(* CODESYS project BUILDING.library
   LanguageModelAttribute: qualified-access-only
   Author: OSCAT
   Version: 1.0.0.1
   Description: OSCAT Library with Building POUs.
      see ww.oscat.de for here home.
   Title: BUILDING
   DefaultNamespace: OSCAT_BUILDING
   Company: OSCAT

Project tree, tasks and I/O mapping:
  libraries: Standard, * (System); BASIC, 3.3.4.0 (OSCAT)
  Data types/
  Global Variables/
    global variables Constants
    global variables Globale_Variablen
    global variables Setup_Data
  POUs/
    actuators/
      function block ACTUATOR_2P [ST]
      function block ACTUATOR_3P [ST]
      function block ACTUATOR_A [ST]
      function block ACTUATOR_COIL [ST]
      function block ACTUATOR_PUMP [ST]
      function block ACTUATOR_UD [ST]
      function block AUTORUN [ST]
    electrical/
      function block CLICK [ST]
      function block CLICK_MODE [ST]
      function block DEBOUNCE [ST]
      function block DIMM_2 [ST]
      function block DIMM_I [ST]
      function block F_LAMP [ST]
      function block PULSE_LENGTH [ST]
      function block PULSE_T [ST]
      function block SW_RECONFIG [ST]
      function block SWITCH_I [ST]
      function block SWITCH_X [ST]
      function block TIMER_1 [ST]
      function block TIMER_2 [ST]
      function TIMER_EVENT_DECODE [ST]
      function block TIMER_EXT [ST]
      function block TIMER_P4 [ST]
    HLK/
      function AIR_DENSITY [ST]
      function AIR_ENTHALPY [ST]
      function block BOILER [ST]
      function block BURNER [ST]
      function DEW_CON [ST]
      function DEW_RH [ST]
      function DEW_TEMP [ST]
      function HEAT_INDEX [ST]
      function block HEAT_METER [ST]
      function block HEAT_TEMP [ST]
      function block LEGIONELLA [ST]
      function SDD [ST]
      function SDD_NH3 [ST]
      function SDT_NH3 [ST]
      function block T_AVG24 [ST]
      function block TANK_LEVEL [ST]
      function TANK_VOL1 [ST]
      function TANK_VOL2 [ST]
      function block TEMP_EXT [ST]
      function WATER_CP [ST]
      function WATER_DENSITY [ST]
      function WATER_ENTHALPY [ST]
      function WCT [ST]
    Jalousie/
      function block BLIND_ACTUATOR [ST]
      function block BLIND_CONTROL [ST]
      function block BLIND_CONTROL_S [ST]
      function block BLIND_INPUT [ST]
      function block BLIND_NIGHT [ST]
      function block BLIND_SCENE [ST]
      function block BLIND_SECURITY [ST]
      function block BLIND_SET [ST]
      function block BLIND_SHADE [ST]
      function block BLIND_SHADE_S [ST]
      function block BLIND_MASTER_CONECTOR [ST]
    Other/
      function BUILDING_VERSION [ST]
  Visualizations/
  global variables PersistentVars
  Documentation/
    oscat-building100-en
    oscat_building100_de
  00000000-0000-0000-0000-000000000000|D:\src\CODESYS Store\OSCAT\OSCAT_Building\trunk\Documents\Documentation\oscat_building100_de.pdf
  00000000-0000-0000-0000-000000000000|C:\Users\e.schwellinger\Desktop\oscat-building100-en.pdf
*)

// Global Variables/Constants
VAR_GLOBAL CONSTANT
END_VAR

// Global Variables/Globale_Variablen
VAR_GLOBAL
END_VAR

// PersistentVars
VAR_GLOBAL PERSISTENT RETAIN
END_VAR

// Global Variables/Setup_Data
VAR_GLOBAL RETAIN

END_VAR

// POUs/actuators/ACTUATOR_2P
FUNCTION_BLOCK ACTUATOR_2P
VAR_INPUT
	IN : BYTE;
	TEST : BOOL;
	ARE : BOOL := TRUE;
END_VAR
VAR_IN_OUT
	ARX : BOOL;
END_VAR
VAR_INPUT CONSTANT
	CYCLE_TIME : TIME;
	SENS : BYTE;
	SELF_ACT_TIME : TIME;
	SELF_ACT_PULSE : TIME;
	SELF_ACT_CYCLES : INT := 1;
END_VAR
VAR_OUTPUT
	OUT : BOOL;
	ARO : BOOL;
END_VAR
VAR
	timer : AUTORUN;
	pwgen : OSCAT_BASIC.GEN_PULSE;
END_VAR


(*
version 2.1	24. jan. 2009
programmer 	hugo
tested by		oscat

this is an intelligent actuator interface for any 2point actuator like coil drive.
the 2Point actuator can only switch on/off and therefore the input must be converted to on/off cycles.
the interface can be programmed with double click on the symbol.
in addition a self_act_time and self_act_cycles ca be programmed to switch n times on/off every self_act_time to avoid a valve to freeze.
the input value must be between 0 and 255. with the setup variable sens one can specify what must be the minimum input to turn the valve on at all.
at the same time an input > 255-sens will turn the valve on at all times.


*)

(* run the autorun timer *)
timer(trun := SELF_ACT_PULSE * (2 * SELF_ACT_CYCLES), toff := SELF_ACT_TIME, Test := TEST, ARE := ARE, arx := ARX);
ARO := timer.ARO;

(* run the pulse width generator *)
IF aro THEN
	pwgen(PTL := SELF_ACT_PULSE, PTH := SELF_ACT_PULSE);
	out := pwgen.Q;
ELSIF in < sens THEN
	out := FALSE;
ELSIF in > BYTE#255 - sens THEN
	out := TRUE;
ELSE
	pwgen.PTH := (CYCLE_TIME * OSCAT_BASIC.BAND_B(IN,SENS)) / 255;
	pwgen.PTL := CYCLE_TIME - pwgen.PTH;
	pwgen();
	out := pwgen.Q;
END_IF;



(* revision history
hm	7.10.2006 		rev 1.1
	changed error pos could not reach 1 or 0 under certain conditions due to error in code.
	changed on and off in force and force_in for better usability.

hm	17.1.2007		rev 1.2
	deleted unused variable time_overflow

hm	15.9.2007		rev 1.3
	replaced time() with T_PLC_MS for compatibility and performance reasons

hm	19. 11 2007		rev 1.4
	replaced left over statement time() with tx

hm	27. 12. 2007	REV 1.5
	CHANGED CODE FOR BETTER PERFORMANCE

hm	21. oct. 2008	rev 1.6
	code optimized

hm	23. nov. 2008	rev 2.0
	new code using library modules

hm	24. jan. 2009	rev 2.1
	deleted unused var inb
*)

END_FUNCTION_BLOCK

// POUs/actuators/AUTORUN
FUNCTION_BLOCK AUTORUN
VAR_INPUT
	IN : BOOL;
	TEST : BOOL;
	ARE : BOOL := TRUE;
END_VAR
VAR_IN_OUT
	ARX : BOOL;
END_VAR
VAR_INPUT CONSTANT
	TRUN : TIME;
	TOFF : TIME;
END_VAR
VAR_OUTPUT
	OUT : BOOL;
	ARO : BOOL;
END_VAR
VAR
	timer : OSCAT_BASIC._RMP_B;
	val : BYTE;
END_VAR



(*
version 1.0	20. nov 2008
programmer 	hugo
tested by	oscat




*)

(* run the integrator when T_off > T#0s *)
IF TOFF > T#0s THEN
	timer(DIR:= OUT, TR := SEL(OUT, TOFF, TRUN), RMP := val);
ELSE
	val := 255;
END_IF;


(* when timer = 0 or test then initiate autorun until timer reaches 255 *)
IF (NOT ARX AND ARE AND val = 0) OR TEST THEN
	val := 0;
	ARO := TRUE;
	ARX := TRUE;
ELSIF val = 255 AND ARO THEN
	ARO := FALSE;
	ARX := FALSE;
END_IF;

(* output is true when autorun ARO is true or in = TRUE *)
out := IN OR ARO;



(* revision history
hm 20. nov. 2008	rev 1.0
	original version

*)

END_FUNCTION_BLOCK

// POUs/electrical/CLICK
FUNCTION_BLOCK CLICK
VAR_INPUT
	in : BOOL;
END_VAR
VAR_OUTPUT
	Q : BOOL;
	single : BOOL;
	double : BOOL;
	triple : BOOL;
	status: BYTE;
END_VAR
VAR_INPUT CONSTANT
	T_debounce : TIME := t#10ms;
	T_short : TIME := t#200ms;
	T_pause : TIME := t#500ms;
	T_reconfig : TIME := t#1m;
END_VAR
VAR
	s_in : SW_RECONFIG;
	tx: TIME;
	state: INT;
	last: TIME;
END_VAR

(*
version 2.0	28. dec. 2008
programmer 	oscat
tested by		oscat

click checks an input for single, double or tripple click and sets the corresponding output single, doulbe or triple for the time the input stays high at the last click.
the maximum high and low time for a click can be configured with setup variables.
the input configures itself to be high or low active depending on which state the input stays longer than t_reconfig.

*)

(* reconfiguration and debounce circuitry *)
s_in(in := in, TD := T_debounce, TR := T_reconfig);

(* read system time *)
tx := DWORD_TO_TIME(OSCAT_BASIC.T_PLC_MS());

(* count the mumber of clicks *)
IF s_in.Q XOR Q THEN
	last := tx;
	IF s_in.Q THEN state := state + 1; END_IF;
END_IF;
Q := s_in.Q;

(* set outputs *)
IF state > 0 THEN
	IF (Q AND tx - last > t_short) OR (NOT Q AND tx - last > t_pause) THEN
		CASE state OF
			1:	single := TRUE;
				status := 111;
			2:	double := TRUE;
				status := 112;
			3:	triple := TRUE;
				status := 113;
		END_CASE;
		state := 0;
	END_IF;
ELSIF NOT q THEN
	single := FALSE;
	double := FALSE;
	triple := FALSE;
	status := 110;
	last := tx;
	state := 0;
END_IF;





(* revision history

15 Feb 2007	rev 1.0	hm
	created original version

18.5.2007	rev 1.1 hm
	corrected an error while execution would stop after t_reconfig elapsed.

15.9.2007	rev 1.2 hm
	replaced Time() with T_PLC_MS for compatibility and performance reasons

28. dec. 2008	rev 2.0
	rewritten using modular approach

*)

END_FUNCTION_BLOCK

// POUs/electrical/DEBOUNCE
FUNCTION_BLOCK DEBOUNCE
VAR_INPUT
	IN : BOOL;
	TD : TIME;
	PM : BOOL;
END_VAR

VAR_OUTPUT
	Q : BOOL;
END_VAR
VAR
	deb : OSCAT_BASIC.TOF;
END_VAR

(*
version 1.0	22. sep. 2008
programmer 	oscat
tested by	tobias

DEBOUNCE is used to debounce switch inputs.
in addition to the debounce functionality this FB can also be used to detect rising edges on IN when PM = TRUE.
When PM = FALSE, Q follows in with the debounce functionality.

*)


IF NOT deb.Q AND IN THEN
	(* rising edge on input detetced a *)
	Q := TRUE;
ELSIF NOT PM THEN
	Q := deb.Q;
ELSE
	Q := FALSE;
END_IF;

(* run debounce timer *)
deb(IN := IN, PT := TD);



(*
hm 22. sep. 2008	rev 1.0
	original version

*)

END_FUNCTION_BLOCK

// POUs/electrical/SW_RECONFIG
FUNCTION_BLOCK SW_RECONFIG
VAR_INPUT
	IN : BOOL;
	TD : TIME;
	TR : TIME;
END_VAR
VAR_OUTPUT
	Q : BOOL;
END_VAR
VAR
	T1, T2 : OSCAT_BASIC.TON;
	INV: BOOL;
END_VAR


(*
version 1.0	22. oct. 2008
programmer 	hugo
tested by	oscat

SW_reconfig detects if an input is high or low active and debounces the input

*)

(* run debounce circuit *)
t1(in := IN, PT := TD);

IF tr > t#0s THEN
	(* generate output *)
	Q := t1.Q XOR inv;
	(* reconfiguration timer *)
	T2(in := Q, pt := TR);
	(* when T2.Q goes high then reverse INV *)
	IF T2.Q THEN INV := NOT INV; END_IF;
ELSE
	Q := t1.Q;
END_IF;



(* revision history
hm	22.10.2008	rev 1.0
	original version

*)

END_FUNCTION_BLOCK

// POUs/actuators/ACTUATOR_3P
FUNCTION_BLOCK ACTUATOR_3P
VAR_INPUT
	IN : BYTE;
	TEST : BOOL;
	ARE : BOOL := TRUE;
	END_POS : BOOL;
END_VAR
VAR_INPUT CONSTANT
	T_RUN : TIME := t#60s;
	T_EXT : TIME := T#10s;
	T_CAL : TIME := t#600s;
	T_DIAG : TIME := T#10d;
	SWITCH_AVAIL : BOOL;
END_VAR
VAR_IN_OUT
	ARX : BOOL;
END_VAR
VAR_OUTPUT
	OUT1 : BOOL;
	OUT2 : BOOL;
	POS : BYTE;
	ERROR : BOOL;
	STATUS : BYTE;
END_VAR
VAR
	ramp : OSCAT_BASIC._RMP_NEXT;
	tx : TIME ;
	next_cal : TIME;
	next_diag : TIME;
	last: TIME;
	start: TIME;
END_VAR


(*
version 2.0	28. jan 2010
programmer 	hugo
tested by		oscat

actuator_3P is an interface for a 3 point actuator.
a 3P actuator is a motor with 2 directions that drives a valve or flap. the position of the valve or flap is controlled by runtime of the motor foreward or backward.
the available inputs are:
IN specifies the position of the actuator, 0 = 0% and 255 = 100%.
an END_POS input is available for an end_pos switch, this switch indicates the valve or flap to be at either 0% or 100%
a TEST input can at any time start a diag cycle which turns the motor towards the 0% position, then measures the runtime to 100% and then the runtime to 0%
these runtimes are stored and used for absolute positioning of the motor during normal operation. this feature is only avaliable with an END_POS switch connected to the input.
a setup variable T_DIAG can be used to specify how often the actuator repeates this auto_diag cycle automatically.
at power on a diag cycle is perfomed automatically.
a time of 0 for T_DIAG means auto diag is never performed.

the outputs out1 and out2 are for the two directions of the motor.
a pos output indicates the simulated position of the actuator during operation.
a error output is activated when the specified max_runtime is reached by any direction during debug without an end_switch to become active.
also when the up and down direction differs by more then 10% the error output is set.

for absolute positioning accuracy the actuator has a setup variable "cal_runtime" if this is set the actuator measures the total runtime of the motors and when this 
cal_runtime is exceeded it resets the actuator to 0% position and sets the output again to assure absolute accuracy.

test and calibration can be shut off by setting the appropriate values to 0.
a switch_available setup variable specifies if end_pos switches are available.

*)

(* read system timer *)
tx := DWORD_TO_TIME(OSCAT_BASIC.T_PLC_MS());

(* check test input *)
IF TEST THEN
	status := 103;
	start := tx;
	ARX := TRUE;
END_IF;

CASE status OF
	0:	(* power on setup *)
		IF ARE AND NOT ARX THEN
			status := 103;
			start := tx;
			ARX := TRUE;
		END_IF;

	100:	(* normal operation *)
		(* check for auto diagnostics *)
		IF T_DIAG > T#0s AND tx > next_diag AND ARE AND NOT ARX THEN
				status := 103;
				start := tx;
				ARX := TRUE;

		(* check for auto calibration *)
		ELSIF T_CAL > T#0s AND tx > next_cal AND ARE AND NOT ARX THEN
			IF pos > BYTE#127 THEN
				OUT1 := TRUE;
				OUT2 := FALSE;
				ramp.IN := 255;
				ARX := TRUE;
			ELSE
				OUT1 := FALSE;
				OUT2 := TRUE;
				ramp.IN := 0;
				ARX := TRUE;
			END_IF;
			status := 101;
			start := tx;
		ELSE
			(* increment next_cal if not active *)
			IF NOT(OUT1 OR OUT2) THEN next_cal := next_cal + (tx-last); END_IF;
			(* set ramp generator to IN *)
			ramp.IN := IN;
		END_IF;

	101:	(* calibrate *)
		IF tx - start < T_EXT THEN
			next_cal := tx + T_CAL;
		ELSIF SWITCH_AVAIL AND END_POS THEN
			STATUS := 100;
			ARX := FALSE;
		ELSIF tx - start > T_EXT + T_RUN THEN
			ERROR := SWITCH_AVAIL;
			ARX := FALSE;
		END_IF;

	103:	(* diagnostics up*)
		(* run up for T_ext *)
		IF tx - start < T_EXT THEN
			ERROR := FALSE;
			ramp.TR := T_RUN;
			ramp.TF := T_RUN;
			OUT1 := TRUE;
			OUT2 := FALSE;
			ramp.IN := 255;
		ELSIF SWITCH_AVAIL AND END_POS THEN
			ramp.TR := tx - start;
			STATUS := 104;
		ELSIF tx - start > T_EXT + T_RUN THEN
			ERROR := SWITCH_AVAIL;
			STATUS := 104;
			start := tx;
		END_IF;

	104:	(* diagnostics dn*)
		IF tx - start < T_ext THEN
			OUT1 := FALSE;
			OUT2 := TRUE;
			ramp.IN := 0;
			next_diag := tx + T_DIAG;
		ELSIF SWITCH_AVAIL AND END_POS THEN
			ramp.TR := tx - start;
			(* check if runtimes differ by more than 10% *)
			IF DINT_TO_TIME(ABS(TIME_TO_DINT(ramp.TR) - TIME_TO_DINT(ramp.TF))*10) > T_RUN THEN error := TRUE; END_IF;
			STATUS := 100;
			ARX := FALSE;
			next_cal := tx + T_CAL;
		ELSIF tx - start > T_EXT + T_RUN THEN
			IF SWITCH_AVAIL THEN ERROR := TRUE; END_IF;
			STATUS := 100;
			ARX := FALSE;
			next_CAL := tx + T_CAL;
		END_IF;
END_CASE;

(* internal flap simulation and output activation *)
ramp(OUT := POS);
IF STATUS = 100 THEN
	OUT1 := ramp.UP;
	OUT2 := ramp.DN;
END_IF;

(* adjust position if end switch is active *)
IF SWITCH_AVAIL AND END_POS THEN
	POS := SEL(POS > 127, 0, 255);
	next_cal := tx + T_CAL;
END_IF;

(* set last to tx for next cycle *)
last := tx;



(* revision history

hm	19. oct 2006	rev 1.1
	added security checks for end_switch to avoid overrun of the end_switch, hans

hm	23. jan 2007	rev 1.2
	deleted unused variables force_on and force_off

hm	15. sep 2007	 rev 1.3
	replaced Time() with T_PLC_MS for compatibility and performance reasons

hm	28. jan 2010	rev 2.0
	new code and new features

*)

END_FUNCTION_BLOCK

// POUs/actuators/ACTUATOR_A
FUNCTION_BLOCK ACTUATOR_A
VAR_INPUT
	I1 : BYTE;
	IS : BOOL;
	I2 : BYTE;
	RV : BOOL;
	DX : BOOL;
END_VAR
VAR_INPUT CONSTANT
	RUNTIME : TIME;
	SELF_ACT_TIME : TIME;
	OUT_MIN : WORD;
	OUT_MAX : WORD;
END_VAR
VAR_OUTPUT
	Y : WORD;
END_VAR
VAR
	timer : OSCAT_BASIC.CYCLE_4;
	dx_edge: BOOL;
END_VAR


(*
version 1.0 8. nov. 2008	
programmer 	hugo
tested by	oscat

ACTUATOR_A drives any valve or similar with 0 - 255 continuous control input.
 
*)

(* run the system timer, if self_act_time = t#0s then state is set to 0 *)
timer(T0 := RUNTIME, T1 := RUNTIME, T3 := SELF_ACT_TIME, sl := DX AND NOT dx_edge, sx := 0, S0 := SELF_ACT_TIME > t#0s);
dx_edge := dx;

CASE timer.STATE OF
	0: 	(* self act min value *)
		Y := OUT_MIN;
	1:	(* self_act max value *)
		Y := OUT_MAX;
	3:	(* normal operation *)
		IF rv THEN
			Y := OUT_MAX - (OUT_MAX - OUT_MIN) * SEL(IS, I1, I2) / 255;
		ELSE
			Y := (OUT_MAX - OUT_MIN) * SEL(IS, I1, I2) / 255 + OUT_MIN;
		END_IF;
END_CASE;




(*
hm 	8. nov. 2008	rev 1.0
	original version

*)

END_FUNCTION_BLOCK

// POUs/actuators/ACTUATOR_COIL
FUNCTION_BLOCK ACTUATOR_COIL
VAR_INPUT
	IN : BOOL;
END_VAR
VAR_INPUT CONSTANT
	self_act_cycle : TIME := t#10d;
	self_act_time : TIME := t#1s;
END_VAR
VAR_OUTPUT
	OUT :BOOL;
	STATUS : BYTE;
END_VAR
VAR
	last : DWORD;
	init: BOOL;
	tx: DWORD;
	now: DWORD;
END_VAR


(*
version 1.0	1. jun. 2008
programmer 	hugo
tested by		tobias

this is an intelligent actuator interface for any coil actuator.
the coil actuator can only switch on/off.
coil actuators like vents can get stuck if they are not u8sed for a long time and need to be autoactivated on ce in a while.

*)

(* read system time *)
now := OSCAT_BASIC.T_PLC_MS();

(* initialize for first cycle *)
IF NOT init THEN
	last := now;
	init := TRUE;
ELSIF IN THEN
	OUT := TRUE;
	STATUS := 101; (* activated by input *)
	LAST := now;
ELSE
	OUT := FALSE;
	STATUS := 100; (* disabled *)
	(* now we need to check for self activation *)
	tx := now - last;
	IF (self_act_cycle > T#0s) AND (tx >= TIME_TO_DWORD(self_act_cycle)) THEN
		OUT := TRUE;
		STATUS := 102; (* auto activation *)
		IF tx >= TIME_TO_DWORD(self_act_cycle + self_act_time) THEN
			last := now;
			OUT := FALSE;
			STATUS := 100; (* idle *)
		END_IF;
	END_IF;
END_IF;



(*
revision history:

hm		1. jun. 2008 	rev 1.0
	original version

*)

END_FUNCTION_BLOCK

// POUs/actuators/ACTUATOR_PUMP
FUNCTION_BLOCK ACTUATOR_PUMP
VAR_INPUT
	IN : BOOL;
	MANUAL : BOOL;
	RST : BOOL;
END_VAR
VAR_INPUT CONSTANT
	MIN_ONTIME : TIME := t#10s;
	MIN_OFFTIME : TIME := t#10s;
	RUN_EVERY : TIME := t#10000m;
END_VAR
VAR_OUTPUT
	PUMP : BOOL;
END_VAR
VAR_IN_OUT
	RUNTIME : UDINT;
	CYCLES : UDINT;
END_VAR
VAR
	tx : TIME;
	last_change : TIME;
	meter : OSCAT_BASIC.ontime;
	old_man : BOOL;
	init: BOOL;
END_VAR

(*
version 1.4		21. oct. 2008
programmer 		oscat
tested BY		oscat

actuator_pump is a pump interface which can be controlled by an input in and an input manual.
in or manual high turns the pump output on.
a rst input is used to reset the runtime counters.
when the pump was not active for a time run_every the actuator turns on the pump automatically for min_ontime.
two setup variables min_ontime and min_offtime guarantee a minimum runtime and offtime of the pump.
the units are hours and the output type is real to prevent from overfow.

*)

tx := DWORD_TO_TIME(OSCAT_BASIC.T_PLC_MS());

IF NOT init THEN
	init := TRUE;
	last_change := tx;
ELSIF rst THEN
	rst := FALSE;
	runtime := 0;
	cycles := 0;
ELSIF manual AND NOT pump AND NOT old_man THEN
	last_change := tx;
	pump := TRUE;
ELSIF NOT manual AND old_man AND pump AND NOT in THEN
	last_change := tx;
	pump := FALSE;
ELSIF in AND NOT pump AND tx - last_change >= min_offtime THEN
	last_change := tx;
	pump := TRUE;
ELSIF pump AND NOT in AND NOT manual AND tx - last_change >= min_ontime THEN
	last_change := tx;
	pump := FALSE;
ELSIF NOT pump AND (tx - last_change >= run_every) AND (run_every > T#0s) THEN
	last_change := tx;
	pump := TRUE;
END_IF;

meter(in := pump, seconds := runtime, cycles := cycles);
old_man := manual;



(*
hm	27.12.2006		rev 1.1
	fixed a failure while the pump would run for tmin after startup.

hm	15.9.2007		rev 1.2
	replaced Time() with T_PLC_MS for compatibility and performance reasons

hm	13. oct. 2008	rev 1.3
	auto activation can now be disabled when run_every = t#0s

hm	21. oct. 2008	rev 1.4
	changed to use ontime rev 2.0

*)

END_FUNCTION_BLOCK

// POUs/actuators/ACTUATOR_UD
FUNCTION_BLOCK ACTUATOR_UD
VAR_INPUT
	UD : BOOL;
	ON : BOOL;
	Manual : BOOL;
	Up : BOOL;
	Dn : BOOL;
	off : BOOL;
	YUP_in : BOOL;
	YDN_in : BOOL;
END_VAR
VAR_INPUT CONSTANT
	TON : TIME;
	TOFF : TIME;
	out_return : BOOL;
END_VAR
VAR_OUTPUT
	Yup : BOOL;
	Ydn : BOOL;
	status : BYTE;
END_VAR
VAR
	tx : TIME;
	last : TIME;
	init: BOOL;
END_VAR

(*
version 1.3	17. oct. 2008
programmer 	hugo
tested by		tobias

out_ud is a up/dn or Right/left locked output driver.
it can be controlled by automatic inputs UD and ON as well as manual inputs for up and dn.
a security input to shut off at any time is prvided by the off input.
two time set inputs ton and toff specify a minimum on time for outputs and a minimum off time before the next output can become active.
the module assures that only one output can be active at any time.
for higher security pls make sure you use hardware locking of the outputs to prevent from defective wiring or outputs.
further security is provided b feedback inputs Yup_in and Ydn_in which are separate inputs for the output signal, if these inputs are not available 
pls connect them directly to Yup and Ydn.
manual mode will override automatic mode by setting the manual input high.
a status output will be 0 for normal operation or 1 - 99 for error reporting and 101 - 199 for status reporting
The status output is ESR comptible.
*)

(* read system time *)
tx := DWORD_TO_TIME(OSCAT_BASIC.T_PLC_MS());

IF NOT init THEN
	(* INITIALIZATION AT FIRST CALL *)
	last := tx;
	init := TRUE;
ELSIF off THEN
	(* emergency shut off detected *)
	Yup := FALSE;
	ydn := FALSE;
	last := tx;
	status := 101;

(* Watch FOR MIN TON TIME *)
ELSIF ((Yup OR Ydn) AND tx - last < Ton) THEN
	RETURN;
ELSIF NOT yup AND NOT ydn AND tx - last < toff THEN
	RETURN;

(* manual operation *)
ELSIF manual THEN
	status := 102;
	(* directional chage set both outs 0 first *)
	IF yup AND NOT up OR ydn AND NOT dn THEN
		ydn := FALSE;
		yup := FALSE;
		last := tx;
	(* manual up operation *)
	ELSIF UP AND NOT DN AND NOT OFF THEN
		Ydn := FALSE;
		Yup := TRUE;
		last := tx;
		status := 103;
	(* manual down operation *)
	ELSIF DN AND NOT UP AND NOT OFF THEN
		Yup := FALSE;
		Ydn := TRUE;
		last := tx;
		status := 104;
	(* maual mode but no up or down *)
	ELSE
		IF YUP OR YDN THEN LAST := tx; END_IF;
		Yup := FALSE;
		ydn := FALSE;
	END_IF;

(* automatic operation *)
ELSE
	(* directional change set outputs low first *)
	IF yup AND NOT ud OR ydn AND UD THEN
		yup := FALSE;
		ydn := FALSE;
		last := tx;
	(* automatic up operation *)
	ELSIF Ud AND on AND NOT OFF THEN
		Ydn := FALSE;
		Yup := TRUE;
		last := tx;
		status := 111;

	(* automatic down operation *)
	ELSIF NOT UD AND on AND NOT OFF THEN
		Yup := FALSE;
		Ydn := TRUE;
		last := tx;
		status := 112;
	(* standby mode *)
	ELSE
		IF Yup OR Ydn THEN last := tx; END_IF;
		Yup := FALSE;
		Ydn := FALSE;
		status := 110;
	END_IF;
END_IF;

(* make sure Yup and Ydn are never on at the same time *)
IF Ydn AND Yup_in AND out_return THEN
	Ydn := FALSE;
	status := 1;
END_IF;
IF Yup AND Ydn_in AND out_return THEN
	Yup := FALSE;
	status := 2;
END_IF;



(* revision history
hm 22. jan 2007	rev 1.1
	added status output
	changed inputs ton, toff to config variables
	added config var out_return to enable yup_in and Ydn_in
	manual mod will override automatic mode 

hm	15.9.2007	rev 1.2
	replaced Time() with T_PLC_MS for compatibility and performance reasons

hm	17. oct. 2008	rev 1.3
	deleted unnecessary initialization with 0
*)

END_FUNCTION_BLOCK

// POUs/HLK/AIR_DENSITY
FUNCTION AIR_DENSITY : REAL
VAR_INPUT
	T : REAL;
	P : REAL;
	RH : REAL;
END_VAR
VAR CONSTANT
	RL : REAL := 287.05;
	RX : REAL := 3.773319E-3;
END_VAR


(*
version 1.3	13. mar. 2009
programmer 	hugo
tested by		tobias

this function calculates the air density between 0 and 100 deg C

*)

AIR_DENSITY := OSCAT_BASIC.phys.PN * (1.0 - RH * SDD(T, TRUE) * RX / P) / (RL * ( T - OSCAT_BASIC.phys.T0));

(* original code used for rev 1.0

SDD := SDD(T,FALSE);
RF := RL / (1- RH*SDD/P*RX);
Air_density := P / (RF * (T-TK));

*)

(* revision history

hm	29.10.2007	rev 1.0
	original version

hm	4.12.2007		rev 1.1
	changed code for better performance

hm	18. oct. 2008	rev 1.2
	using phys constants

hm	13. mar. 2009	rev 1.3
	real constants updated to new systax using dot

*)

END_FUNCTION

// POUs/HLK/SDD
FUNCTION SDD : REAL
VAR_INPUT
	T : REAL;
	ICE: BOOL;
END_VAR


(*
version 1.1	2 dec 2007
programmer 	hugo
tested by		tobias

this function calculates the vapor saturation pressure for moist Air over ice or water

*)

IF ice THEN
	SDD := 611.153 * EXP(22.4433 * T / (272.186 + T));
ELSE
	SDD := 611.213 * EXP(17.5043 * T / (241.2 + T));
END_IF;



(* revision history

hm 29 oct 2007		rev 1.0
	original version

hm	2. dec 2007		rev 1.1
	changed code for better performance
*)

END_FUNCTION

// POUs/HLK/AIR_ENTHALPY
FUNCTION AIR_ENTHALPY : REAL
VAR_INPUT
	T : REAL;
	RH : REAL;
END_VAR
VAR CONSTANT
	CPL : REAL := 1.00482;
	CW : REAL := 1.86;
	LH : REAL := 2500.78;
END_VAR


(*
version 1.1	2 nov 2007
programmer 	hugo
tested by		tobias

this function calculates the enthalpy for humid air between 0 and 100 deg C

*)

AIR_ENTHALPY := CPL * T + (CW * T + LH) * DEW_CON(RH,T);

(* revision history

hm	31.10.2007	rev 1.0
	original version

hm	2.11.2007		rev 1.1
	deleted unused variable RF

hm	2.12.2007		rev 1.2
	changed code for better performance
*)

END_FUNCTION

// POUs/HLK/DEW_CON
FUNCTION DEW_CON : REAL
VAR_INPUT
	RH : REAL;
	T : REAL;
END_VAR


(*
version 1.6	19. jan. 2011
programmer 	hugo
tested by		oscat

this function calculates the water concentratin in air for a given temperature and relative humidity.
the output states the concentration of water vapor in air in Gramms / qubic meter.

*)

(*	this code is good to read but need to be improoved
	SDD := 6.1078*EXPT(10,(a*T)/(b+T));
	DD := RH/100 * SDD;
	V := LOG(DD/6.1078);
	TD := b*V/(a-v);
	dew_con := 0.1 * mw / RU * DD / (T - TK);
*)
IF RH > 0.0 AND T > -50.0 THEN
	DEW_CON := 2.166824303E-2 * RH * SDD(T,FALSE)  / (T - OSCAT_BASIC.phys.T0);
ELSE
	DEW_CON := 0.0;
END_IF;

(*
Bezeichnungen:
r = relative Luftfeuchte
T = Temperatur in °C
TK = Temperatur in Kelvin (TK = T + 273.15)
TD = Taupunkttemperatur in °C
DD = Dampfdruck in hPa
SDD = Sättigungsdampfdruck in hPa

Parameter:
a = 7.5, b = 237.3 für T >= 0
a = 7.6, b = 240.7 für T < 0 über Wasser (Taupunkt)
a = 9.5, b = 265.5 für T < 0 über Eis (Frostpunkt)

R* = 8314.3 J/(kmol*K) (universelle Gaskonstante)
mw = 18.016 kg (Molekulargewicht des Wasserdampfes)
AF = absolute Feuchte in g Wasserdampf pro m3 Luft

Formeln:

   1. SDD(T) = 6.1078 * 10^((a*T)/(b+T))
   2. DD(r,T) = r/100 * SDD(T)
   3. r(T,TD) = 100 * SDD(TD) / SDD(T)
   4. TD(r,T) = b*v/(a-v) mit v(r,T) = log10(DD(r,T)/6.1078)
   5. AF(r,TK) = 10^5 * mw/R* * DD(r,T)/TK; AF(TD,TK) = 10^5 * mw/R* * SDD(TD)/TK 

*)

(* revision history

hm 29 apr 2007	rev 1.0
	original version

hm	13.sep 2007	rev 1.1
	improoved coding for speed
	deleted unused variabled SDD,DD,V, TD

hm	2. dec 2007	rev 1.2
	changed code for better performance
	output is now in Gramms / Qubic meter

hm	14. oct. 2008	rev 1.3
	performance improvement

hm	18. oct. 2008	rev 1.4
	using phys constants

hm	13. mar. 2009	rev 1.5
	improved code

hm	19. jan. 2011	rev 1.6
	return value 0.0 if RH <= 0.0

*)

END_FUNCTION

// POUs/Jalousie/BLIND_ACTUATOR
 FUNCTION_BLOCK BLIND_ACTUATOR
VAR_INPUT
	UP, DN : BOOL;
	S_IN : BYTE;
	T_UD : TIME := T#10s;
	T_ANGLE : TIME := T#3s;
END_VAR
VAR_INPUT CONSTANT
	T_LOCKOUT : TIME := t#100ms;
END_VAR
VAR_OUTPUT
	POS, ANG : BYTE;
	QU, QD : BOOL;
	STATUS : BYTE;
END_VAR
VAR
	position, angle : OSCAT_BASIC.RMP_B;
	lock : OSCAT_BASIC.INTERLOCK;
END_VAR

(*
version 1.4	08. mar. 2010
programmer 	AE
tested by	AE


blind actuator drives the up and down motor of a blind. T_lockout specifies the time between up or dn becomes active. 
To change direction there must be a minimum wait time to allow the motors to come to rest first.
the up and down outputs QU and QD are controlled by the inputs UP and DN.
the outputs pos and ang simulate the position of the blind pos = 0 means blind is down and pos = 255 = blind is up.
the angle 0 means vertical posisition of the slates and 255 means horizontal position of the slates.


*)

(* make sure only one motor is active at a given time *)
lock(i1 := UP, I2 := DN, TL := T_lockout);

(* ramp up or down to simulate the angle position of the blind slats *)
angle(e := lock.Q1 OR lock.Q2, UP := lock.Q1, PT := T_Angle);
position(e := lock.Q1 AND angle.high OR lock.Q2 AND angle.low, up := lock.Q1, PT := T_UD);

(* set the outputs *)
pos := position.Out;
ang := angle.Out;

(* set the outputs *)
QU := lock.Q1;
QD := lock.Q2;

(* set the status output *)
IF UP AND DN THEN
	 status := 1;			(* error up and down together are not allowed *)
ELSIF UP THEN
	status := 121;
ELSIF DN THEN
	status := 122;
ELSE
	status := S_IN;
END_IF;


(* revision history
hm	29. sep 2007	rev 1.0
	original release

hm	6. oct 2007	rev 1.1
	rearanged outputs

hm	18. oct. 2008	rev 1.2
	changed calls for rmp_B because of change in RMP_B

hm	27. jul. 2009	rev 1.3
	changes status to be 12X

ae	08. mar. 2010 rev 1.4	
	at aPosition

*)

END_FUNCTION_BLOCK

// POUs/Jalousie/BLIND_CONTROL
FUNCTION_BLOCK BLIND_CONTROL
VAR_INPUT
	UP, DN : BOOL;
	S_IN : BYTE;
	PI : BYTE;
	AI : BYTE;
	T_UD, T_ANGLE : TIME;
END_VAR
VAR_INPUT CONSTANT
	SENS : BYTE := 5;
	T_LOCKOUT: TIME := T#100ms;
END_VAR
VAR_OUTPUT
	POS, ANG : BYTE;
	MU, MD : BOOL;
	STATUS : BYTE;
END_VAR
VAR
	act : BLIND_ACTUATOR;
	delta : BYTE;
	bTimeTest:BOOL:=FALSE;
	iPos:BYTE;
	iAngel:BYTE;
END_VAR

(*
version 1.5		8. mar 2011
programmer 		AE
tested by		AE

*)

IF bTimeTest THEN
	PI:=iPos;
	AI:=iAngel;
	UP:=TRUE;
	DN:=TRUE;
END_IF

(* Check Position*)
act(T_UD:=T_UD, T_ANGLE:=T_ANGLE, T_lockout := T_Lockout);

IF UP AND DN THEN
	(* automatic modus detected *)
	(* first find correct position *)
	IF BYTE_TO_INT(act.pos) < BYTE_TO_INT(pi) - delta THEN
		act.UP := TRUE;
		act.DN := FALSE;
		delta := 0;
		STATUS := 121;
	ELSIF BYTE_TO_INT(act.pos) > BYTE_TO_INT(pi) + delta THEN
		act.UP := FALSE;
		act.DN := TRUE;
		delta := 0;
		STATUS := 122;
	(* regulate angle *)
	ELSIF BYTE_TO_INT(act.ang) < BYTE_TO_INT(ai) - delta AND T_angle > T#100ms THEN
		act.UP := TRUE;
		act.DN := FALSE;
		delta := sens/2;
		STATUS := 123;
	ELSIF BYTE_TO_INT(act.ang) > BYTE_TO_INT(ai) + delta AND T_angle > T#100ms THEN
		act.UP := FALSE;
		act.DN := TRUE;
		delta := sens/2;
		STATUS := 124;
	(* correct position reached *)
	ELSE
		act.UP := FALSE;
		act.DN := FALSE;
		delta := sens;
		STATUS := S_IN;
	END_IF;
ELSE
	act.UP := UP;
	act.DN := DN;
	STATUS := S_IN;
END_IF;

(* blind control calls blind_actuator *)
act(T_UD:=T_UD, T_ANGLE:=T_ANGLE, T_lockout := T_Lockout);
pos := act.pos;
ang := act.ang;
MU := act.QU;
md := act.QD;
status := act.status;

(* revision history
hm	29. sep 2007	rev 1.0
	original release

hm	6. oct 2007	rev 1.1
	rearranged outputs
	integrated blind_actuator into blind_control

hm	16. oct 2007	rev 1.2
	ignore angle when t_angle = 0

hm 29. oct 2007	rev 1.3
	added lockout configuration time for motor direction change
	sens has a setup value of 5

hm	27. jul. 2009	rev 1.4
	changed status handling

ae	08. mar. 2010	rev 1.5
	at aPosition bevor control
	at tolerance "delta := sens/2;"

*)

END_FUNCTION_BLOCK

// POUs/Jalousie/BLIND_CONTROL_S
FUNCTION_BLOCK BLIND_CONTROL_S
VAR_INPUT
	UP, DN : BOOL;
	S_IN : BYTE := 125;
	PI : BYTE;
	T_UP : TIME;
	T_DN : TIME;
	RU : BOOL;
	RD : BOOL;
END_VAR
VAR_INPUT CONSTANT
	T_LOCKOUT: TIME := T#100ms;
	T_EXT : TIME;
	EXT_TRIG : BYTE := 5;
	R_POS_TOP : BYTE := 255;
	R_POS_BOT : BYTE;
END_VAR
VAR_OUTPUT
	POS : BYTE;
	MU, MD : BOOL;
	STATUS : BYTE;
END_VAR
VAR
	rmp : OSCAT_BASIC._RMP_NEXT;
	tx, last : TIME;
	PI_last: BYTE;
END_VAR


(*
version 1.2	23. jan 2010
programmer 	hugo
tested by		heinz


*)


(* status definition
	121 = manual up				manual up operation UP = true and DN = false
	122 = manual down			manual down operation DN = true and UP = false
	123 = auto positioning		automatic mode DN = UP = TRUE
	124 = revert					revert from top or bottom
	125 = nothing					default input for S_IN
	127 = Lockout time			lockout between directional change
	128 = calibrate				calibrate after power up
	129 = extend					extend runtime at top or bottom for continuous calibration
*)

(* read system time *)
tx := DWORD_TO_TIME(OSCAT_BASIC.T_PLC_MS());

(* check inputs and start state machine *)
IF UP  AND NOT DN THEN
	(*  manual UP *)
	rmp.IN := 255;
	STATUS := 121;
ELSIF DN AND NOT UP THEN
	(* manual DN *)
	rmp.IN := 0;
	STATUS := 122;
ELSIF NOT (UP OR DN) THEN
	(* manual standby mode *)
	rmp.IN := PI;
	STATUS := S_IN;
END_IF;

(* simulate pos output *)
rmp(E := UP OR DN, TR := T_UP, TF := T_DN, TL := T_LOCKOUT, OUT := POS);

(* state machine *)
CASE STATUS OF
	0:		(* power up init *)
		last := tx;
		PI_last := PI XOR BYTE#255;
		STATUS := 128;		(* calibrate *)

	121: 	(* manual up *)
		MU := TRUE;
		MD := FALSE;
		IF POS >= (BYTE#255 - EXT_TRIG) THEN
			(* extend cycle if top is reached *)
			POS := 255;
			last := tx;
			STATUS := 129;	(* extend *)
		END_IF;

	122:	(* manual down *)
		MD := TRUE;
		MU := FALSE;
		IF POS <= EXT_TRIG THEN
			(* extend cycle if bottom is reached *)
			POS := 0;
			last := tx;
			STATUS := 129;	(* extend *)
		END_IF;

	123:	(* auto positioning *)
		MD := rmp.DN;
		MU := rmp.UP;
		IF NOT (rmp.DN OR rmp.UP) THEN
			(* automatic position is reached *)
			IF POS <= EXT_TRIG THEN
				(* extend at bottom *)
				MD := TRUE;
				last := tx;
				STATUS := 129;	(* extend *)
			ELSIF POS >= (BYTE#255 - EXT_TRIG)  THEN
				(* extend at top *)
				MU := TRUE;
				last := tx;
				STATUS := 129;	(* extend *)
			ELSE
				STATUS := S_IN;
			END_IF;
		END_IF;

	124:	(* revert from top or bottom *)
		MD := rmp.DN;
		MU := rmp.UP;
		IF NOT(rmp.DN OR rmp.UP) THEN
(*		IF POS = rmp.IN THEN  *)
			PI_last := PI;
			STATUS := S_IN;
		END_IF;

	127:	(* lockout time *)
		IF (tx - last) >= T_LOCKOUT THEN
				STATUS := S_IN;
		END_IF;

	128:	(* calibration *)
		MU := TRUE;
		MD := FALSE;
		rmp.IN := 255;
		IF (tx - last) >= (T_UP +  T_EXT) THEN
			MU := FALSE;
			last := tx;
			STATUS := 127;	(* lockout *)
		END_IF;

	129: (* extend mode *)
		IF (tx - last) >= T_EXT THEN
			MU := FALSE;
			MD := FALSE;
			last := tx;
			STATUS := 127;	(* lockout *)
		END_IF;

ELSE
	MU := FALSE;
	MD := FALSE;
	IF PI <> PI_last THEN
		PI_last := PI;
		rmp.IN := PI;
		STATUS := 123;	(* auto positioning *)
	ELSIF POS = 0 AND RU THEN
		rmp.IN := R_POS_BOT;
		STATUS := 124;	(* revert *)
	ELSIF pos = 255 AND RD THEN
		rmp.IN := R_POS_TOP;
		STATUS := 124;	(* revert *)
	ELSE
		STATUS := S_IN;
	END_IF;
END_CASE;



(* revision history

hm	9. mar. 2009	rev 1.0
	original release

hf	27. jul 2009	rev 1.1
	major code changes and updates

hf	23. Jan 2010	rev 1.2
	fixed a bug during calibration
	added T_UP and T_DN

*)

END_FUNCTION_BLOCK

// POUs/Jalousie/BLIND_INPUT
FUNCTION_BLOCK BLIND_INPUT
VAR_INPUT
	UP, DN: BOOL;
	POS, ANG : BYTE;
	S1, S2 : BOOL;
	IN : BOOL;
	PI, AI : BYTE;
	//S_IN:BYTE := 250;

END_VAR
VAR_INPUT CONSTANT
	SINGLE_SWITCH : BOOL;
	CLICK_EN : BOOL := TRUE;
	CLICK_TIME : TIME := T#500ms;
	MAX_RUNTIME : TIME := T#60s;
	MANUAL_TIMEOUT: TIME := T#1h;
	DEBOUNCE_TIME : TIME := T#20ms;
	DBL_CLK1 : BOOL := FALSE;
	DBL_POS1 : BYTE;
	DBL_ANG1 : BYTE;
	DBL_CLK2 : BOOL := FALSE;
	DBL_POS2 : BYTE := 255;
	DBL_ANG2 : BYTE := 255;
	D1_TOGGLE : BOOL := TRUE;
	D2_TOGGLE : BOOL := TRUE;
	MASTER_MODE : BOOL;
	NO_AUTO_AUTO: BOOL := FALSE;
END_VAR
VAR_OUTPUT
	QU : BOOL := TRUE;
	QD : BOOL := TRUE;
	STATUS : BYTE;
	PO : BYTE := 255;
	AO : BYTE := 255;
	D1, D2 : BOOL;
END_VAR
VAR
	s1e, s2e : OSCAT_BASIC.TOF;
	s1d, s2d : CLICK_MODE;
	dir : BOOL;
	tx, last : TIME;
	R1, R2:Standard.R_TRIG;
	startupDone: BOOL;

END_VAR

(*
version 1.7	12. nov. 2009
programmer 	hugo
tested by		oscat


*)

(* read system timer *)
tx := DWORD_TO_TIME(OSCAT_BASIC.T_PLC_MS());

(* inputs S1 and S2 are debounced and then decoded for multiple clicks *)
s1e(in := S1, pt := DEBOUNCE_TIME);
s2e(in := S2, pt := DEBOUNCE_TIME);
s1d(in := (s1e.Q AND NOT SINGLE_SWITCH) OR (s1e.Q AND SINGLE_SWITCH AND dir), t_long := CLICK_TIME);
s2d(in := (s2e.Q AND NOT SINGLE_SWITCH) OR (s1e.Q AND SINGLE_SWITCH AND NOT dir), t_long := CLICK_TIME);

(* if d1 and d2 are not toggle clear them to make sure they are only active for oine cycle *)
IF NOT d1_toggle THEN d1 := FALSE; END_IF;
IF NOT d2_toggle THEN d2 := FALSE; END_IF;

(* decode actions *)
IF (s1d.LONG AND s2d.LONG) OR (status = 139) THEN
   status := 139;
   IF NOT (s1d.LONG OR s2d.LONG)  THEN status := 130; END_IF;
ELSIF s1d.tp_LONG THEN
	status := 132;
ELSIF s2d.tp_LONG THEN
	status := 133;
ELSIF  s1d.SINGLE THEN
	IF click_en THEN
		(* if running then we stop otherwise start new direction *)
		IF QU XOR QD THEN
			status := 131;
		ELSE
			status := 134;
			last := tx;
			dir := NOT dir;
		END_IF;
	END_IF;
ELSIF  s2d.SINGLE THEN
	IF click_en THEN
		(* if running then we stop otherwise start new direction *)
		IF QU XOR QD THEN
			status := 131;
		ELSE
			status := 135;
			last := tx;
			dir := NOT dir;
		END_IF;
	END_IF;
ELSIF in THEN
	status := 136;
	last := tx;
ELSIF s1d.DOUBLE THEN
	IF dbl_clk1 THEN
		(* a position need to be set for a double click on S1 *)
		status := 137;
		last := tx;
	ELSE
		(* toggle the output when dbl_clk1 is not active *)
		D1 := NOT D1;
	END_IF;
ELSIF s2d.DOUBLE THEN
	IF dbl_clk2 THEN
		(* a position need to be set for a double click on S2 *)
		status := 138;
		last := tx;
	ELSE
		(* toggle the output when dbl_clk2 is not active *)
		(* in single switch mode we need to toggle d1 instead of d2 *)
		IF single_switch THEN D1 := NOT D1; ELSE D2 := NOT D2; END_IF;
	END_IF;
END_IF;
R1(CLK:= DN);
R2(CLK:= UP);
IF R1.Q OR R2.Q THEN
	status := 130;
	startupDone := TRUE;
END_IF 

(* state machine *)
CASE status OF
	0:		(* power up operation *)
			IF NO_AUTO_AUTO THEN
				status := 131;
			ELSE
				status := 130;
			END_IF
			

	130:	(* automatic operation standby *)
			IF NOT master_mode THEN
				PO := POS;
				AO := ANG;
			END_IF;  
			IF NOT NO_AUTO_AUTO OR NOT startupDone THEN
				QU := TRUE;
				QD := TRUE;
			ELSE
				QU := UP;
				QD := DN;
			END_IF

	131:	(* manual operation standby *)
			QU := FALSE;
			QD := FALSE;
			PO := POS;
			AO := ANG;
			(* manual mode will be ended when timeout is reached *)
			IF (tx - last >= manual_timeout) AND NOT NO_AUTO_AUTO THEN
				status := 130;
			END_IF;

	132:	(* manual operation up *)
			QU := TRUE;
			QD := FALSE;
			PO := POS; AO := ANG;
			last := tx;
			IF NOT s1d.LONG THEN status := 131; dir := NOT dir; END_IF;

	133:	(* manual operation down *)
			QU := FALSE;
			QD := TRUE;
			PO := POS; AO := ANG;
			last := tx;
			IF NOT s2d.LONG THEN	status := 131; dir := NOT dir; END_IF;

	134:	(* manual operation single click up *)
			QU := TRUE;
			QD := FALSE;
			PO := POS; AO := ANG;
			IF tx - last >= max_runtime THEN status := 131; END_IF;

	135:	(* manual operation single click dn *)
			QU := FALSE;
			QD := TRUE;
			PO := POS; AO := ANG;
			IF tx - last >= max_runtime THEN status := 131;	END_IF;

	136:	(* forced input in = true *)
			QU := TRUE;
			QD := TRUE;
			PO := PI; AO := AI;
			IF tx-last >= max_runtime THEN status := 130; END_IF;

	137:	(* double click1 position *)
			QU := TRUE;
			QD := TRUE;
			PO := DBL_POS1;
			AO := DBL_ANG1;
			IF tx - last >= max_runtime THEN status := 131; END_IF;

	138:	(* double click2 position *)
			QU := TRUE;
			QD := TRUE;
			PO := DBL_POS2;
			AO := DBL_ANG2;
			IF tx - last >= max_runtime THEN status := 131; END_IF;

	   139:   (* manual operation standby *)
	         QU := FALSE;
	         QD := FALSE;
	         PO := POS;
	         AO := ANG;

END_CASE;


(* revision history
hm	29. sep 2007	rev 1.0
	original release

hm	6. oct 2007		rev 1.1
	renamed ps and as to po and ao

hm	30. dec 2007	rev 1.2
	added click_timeout variable and function

hm	16. jul. 2008	rev 1.3
	rewirtten code to allow for more functionality
	added single click mode with single_switch.
	added Debounce for inputs S1 and S2
	added double_click functionality

hm	26. sep. 2008	rev 1.4
	corrected an error while POS and ANG was transferred to outputs PO and AO during automatic modes

hm	22. jan 2009	rev 1.5
	added pulse mode for double click outputs
	added automatic mode for IN

hm	27. jul 2009	rev 1.6
	changed status 0 to 130

HF	12. nov. 2009	rev 1.7
	added state 139
	set defaults for QU, QD, PO

*)

END_FUNCTION_BLOCK

// POUs/electrical/CLICK_MODE
FUNCTION_BLOCK CLICK_MODE
VAR_INPUT
	IN : BOOL;
END_VAR
VAR_OUTPUT
	SINGLE : BOOL;
	DOUBLE : BOOL;
	LONG : BOOL;
	TP_LONG : BOOL;
END_VAR
VAR_INPUT CONSTANT
	T_LONG : TIME := t#500ms;
END_VAR
VAR
	Timer : OSCAT_BASIC.TP;
	cnt : INT;
	last : BOOL;
END_VAR


(*
version 1.0	13. nov. 2008
programmer 	oscat
tested by	hugo

click_mode decodes an input for single, double or long click and sets the corresponding output single, doulbe or long.
the input configures itself to be high or low active depending on which state the input stays longer than t_reconfig.

*)

(* when input goes high start the timer to decode pulses *)
timer(in := IN, PT := T_LONG);
single := FALSE;
double := FALSE;

IF timer.Q THEN
	(* decode pulses while the timer is active *)
	IF NOT in AND last THEN	cnt := cnt + 1; END_IF;
ELSE
	CASE cnt OF
		1 : single := TRUE;
		2 : double := TRUE;
	END_CASE;
	cnt := 0;
END_IF;
last := in;
TP_LONG := NOT timer.Q AND (NOT LONG) AND IN;
LONG := NOT timer.Q AND in;




(* revision history

hm	13. nov. 2008	rev 1.0
	original release

*)

END_FUNCTION_BLOCK

// POUs/Jalousie/BLIND_NIGHT
FUNCTION_BLOCK BLIND_NIGHT
VAR_INPUT
	UP, DN : BOOL;
	S_IN : BYTE;
	PI, AI : BYTE;
	E_NIGHT : BOOL := TRUE;
	E_DAY	: BOOL := TRUE;
	DTIN : DT;
	SUNRISE, SUNSET : TOD;
END_VAR
VAR_INPUT CONSTANT
	SUNRISE_OFFSET : TIME;
	SUNSET_OFFSET : TIME;
	NIGHT_POSITION : BYTE;
	NIGHT_ANGLE : BYTE;
END_VAR
VAR_OUTPUT
	QU, QD : BOOL;
	STATUS : BYTE;
	PO, AO : BYTE;
END_VAR
VAR
	night : BOOL;
	last_night, last_day : DATE;
END_VAR

(*
version 1.2	6 oct 2007
programmer 	hugo
tested by		tobias


*)

IF NOT (up AND dn) AND night THEN
	(* manual operation at night will cancel operation for one night *)
	night := FALSE;
ELSIF (DT_TO_TOD(dtin) > sunset + sunset_offset) AND (last_night < DT_TO_DATE(dtin)) AND NOT night AND e_night THEN
	(* enable night *)
	night := TRUE;
	last_night := DT_TO_DATE(dtin);
ELSIF (DT_TO_TOD(dtin) > sunrise + sunrise_offset) AND (last_day < DT_TO_DATE(dtin)) AND night AND e_day AND (last_night < DT_TO_DATE(dtin)) THEN
	(* disable night *)
	night := FALSE;
	last_day := DT_TO_DATE(dtin);
END_IF;

(* shade at night only in auto mode and enable = true *)
IF UP AND DN AND night THEN
	status := 141;
	po := night_position;
	ao := night_angle;
ELSE
	QU := UP;
	QD := DN;
	po := pi;
	ao := ai;
	status := s_in;
END_IF;


(* revision history
hm	29. sep 2007	rev 1.0
	original version

hm	5. oct 2007		rev 1.1
	added enable input

hm	6. oct 2007		rev 1.2
	added pos and angle inputs and outputs
	night position and angle can now be configured
	any manual operation at night will cancel night operation

*)

END_FUNCTION_BLOCK

// POUs/Jalousie/BLIND_SCENE
FUNCTION_BLOCK BLIND_SCENE
VAR_INPUT
	UP, DN : BOOL;
	S_IN : BYTE;
	PI, AI : BYTE;
	ENABLE : BOOL;
	SWRITE : BOOL;
	SCENE : BYTE;
END_VAR
VAR_OUTPUT
	QU, QD : BOOL;
	STATUS : BYTE;
	PO, AO : BYTE;
END_VAR
VAR RETAIN
	sx : ARRAY[0..15,0..2] OF BYTE;
END_VAR
VAR_TEMP
	x : BYTE;
END_VAR

(*
version 1.1	29. jan 2008
programmer 	hugo
tested by		tobias


*)

(* delete all bits except the lower 4 of scene *)
x := scene AND 16#0F;

IF enable AND sx[x,2] > 0 AND UP AND DN THEN
	po := sx[x,0];
	ao := sx[x,1];
	status := 160 + x;  (* Status number is 160 to 175 for the 16 scenes *)
	QU := TRUE;
	QD := TRUE;
ELSE
	QU := UP;
	QD := DN;
	status := S_IN;
	po := pi;
	ao := ai;
END_IF;

(* write scene if necessary *)
IF swrite THEN
	status := 176;		(* write scene *)
	sx[x,0] := pi;
	sx[x,1] := ai;
	IF enable THEN sx[x,2] := 1; ELSE sx[x,2] := 0; END_IF; (* if sx[x,2] = 0 the scene is disabled *)
END_IF;


(* revision history
hm	24. oct 2007	rev 1.0
	original release

hm		29.1.2008	rev 1.1
	replaced shr/shl with and for better performance
*)

END_FUNCTION_BLOCK

// POUs/Jalousie/BLIND_SECURITY
FUNCTION_BLOCK BLIND_SECURITY
VAR_INPUT
	UP, DN : BOOL;
	S_IN : BYTE;
	PI, AI : BYTE;
	FIRE : BOOL;
	WIND : BOOL;
	ALARM : BOOL;
	DOOR : BOOL;
	RAIN : BOOL;
END_VAR
VAR_INPUT CONSTANT
	Alarm_UP : BOOL := TRUE;
	WIND_UP :BOOL := TRUE;
	RAIN_UP : BOOL := FALSE;
END_VAR
VAR_OUTPUT
	QU, QD : BOOL;
	STATUS : BYTE;
	PO, AO : BYTE;
END_VAR


(*
version 1.2	12. feb 2008
programmer 	hugo
tested by		tobias


*)

IF Fire THEN
	QU := TRUE;
	QD := FALSE;
	status := 111;
ELSIF Wind THEN
	QU := Wind_up;
	QD := NOT wind_up;
	status := 112;
ELSIF alarm THEN
	QU := Alarm_up;
	QD := NOT Alarm_up;
	status := 113;
ELSIF Door THEN
	QU := TRUE;
	QD := FALSE;
	status := 114;
ELSIF Rain AND NOT (up XOR dn) THEN
	QU := rain_up;
	QD := NOT rain_up;
	status := 115;
ELSE
	QU := UP;
	QD := DN;
	status := S_IN;
	po := pi;
	ao := ai;
END_IF;


(* revision history
hm	29. sep 2007	rev 1.0
	original release

hm	6. oct 2007		rev 1.1
	added pos and angle inputs and outputs
	manual will override rain position
	alarm position can now be configured

hm		12. feb. 2008	rev 1.2
	added config variables rain_up and wind_up
	position for rain and wind is now configurable
*)

END_FUNCTION_BLOCK

// POUs/Jalousie/BLIND_SET
FUNCTION_BLOCK BLIND_SET
VAR_INPUT
	UP, DN : BOOL;
	S_IN : BYTE;
	PI, AI : BYTE;
	IN : BOOL;
	PX, AX : BYTE;
END_VAR
VAR_INPUT CONSTANT
	OVERRIDE_MANUAL : BOOL;
	RESTORE_POSITION : BOOL;
	RESTORE_TIME : TIME := T#60s;
END_VAR
VAR_OUTPUT
	QU, QD : BOOL;
	STATUS : BYTE;
	PO, AO : BYTE;
END_VAR
VAR
	tx: TIME;
	ps: BYTE;
	as: BYTE;
	last: TIME;
END_VAR

(*
version 1.0	27. jul 2009
programmer 	hugo
tested by		oscat

BLIND_SET can be used to force a definite position and angle.
blind_set can be placed close to blind_control for high priority while blind_input must be always at the beginning of the chain with low priority.

*)

(* read system time *)
tx := DWORD_TO_TIME(OSCAT_BASIC.T_PLC_MS());

(* check inputs *)
IF IN THEN
	IF override_manual OR (UP AND DN) THEN
		status := 178;
	END_IF;
END_IF;

(* state machine *)
CASE STATUS OF
	0: (* power on state *)
		status := S_IN;

	178: (* force values from PX and AX *)
		PO := PX;
		AO := AX;
		QU := TRUE;
		QD := TRUE;
		(* check for end of forced position *)
		IF NOT in THEN
			STATUS := SEL(RESTORE_POSITION, S_IN, 179);
			last := tx;
		END_IF;

	179: (* restore previous position *)
		PO := ps;
		AO := as;
		IF ((PO = PI) AND (AO = AI))  OR tx - last >= RESTORE_TIME THEN
			status := S_IN;
		END_IF;

ELSE
	(* no operation transfer inputs to outputs *)
	PO := PI;
	ps := PI;
	AO := AI;
	as := AI;
	STATUS := S_IN;
	QU := UP;
	QD := DN;
END_CASE;


(* revision history
hm	27. jul 2009	rev 1.0
	original release

*)

END_FUNCTION_BLOCK

// POUs/Jalousie/BLIND_SHADE
FUNCTION_BLOCK BLIND_SHADE
VAR_INPUT
	UP, DN : BOOL;
	S_IN : BYTE;
	PI, AI : BYTE;
	ENABLE : BOOL;
	SUN : BOOL;
END_VAR
VAR_IN_OUT
	CX : OSCAT_BASIC.CALENDAR;
END_VAR
VAR_INPUT CONSTANT
	sunrise_offset : TIME := T#1h;
	sunset_preset : TIME := T#1h;
	direction : REAL := 180.0;
	angle_offset : REAL := 80.0;
	slat_width : REAL := 80.0;
	Slat_spacing : REAL := 60.0;
	Shade_delay : TIME := T#60s;
	Shade_pos : BYTE;
END_VAR
VAR_OUTPUT
	QU, QD : BOOL;
	STATUS : BYTE;
	PO, AO : BYTE;
END_VAR
VAR
	angle: REAL;
	sun_delay : OSCAT_BASIC.TOF;
END_VAR

(*
version 1.4	13. mar. 2009
programmer 	hugo
tested by		tobias


*)

(* the input sun is sent through tof which will delay the shade for the time shade_delay *)
sun_delay(IN := sun, PT := shade_delay);

IF UP AND DN AND enable AND sun_delay.Q AND cx.SUN_HOR > direction - angle_offset AND cx.SUN_HOR < direction + angle_offset AND
	DT_TO_TOD(cx.UTC) > cx.SUN_RISE + sunrise_offset AND DT_TO_TOD(cx.UTC) < cx.SUN_SET - sunset_preset THEN
	status := 151;
	QU := UP;
	QD := DN;
	(* position is predefined *)
	po := shade_pos;
	(* shading is active now calculate the slat angle *)
	(* calculate the max angle for the blind *)
	angle := OSCAT_BASIC.DEG(ATAN(slat_spacing / slat_width));
	(* check if sun angle is between 0 and max angle *)
	IF cx.SUN_VER > 0.0 AND cx.SUN_VER < angle THEN
		angle := cx.SUN_VER + OSCAT_BASIC.DEG(ACOS(COS(OSCAT_BASIC.RAD(cx.SUN_VER))*slat_spacing / Slat_width));
		ao := INT_TO_BYTE(DINT_TO_INT(LIMIT(0,TRUNC(angle * 2.833333333), 255)));
	ELSE
		ao := 255;
	END_IF;
ELSE
	QU := UP;
	QD := DN;
	po := pi;
	ao := ai;
	status := S_IN;
END_IF;

(* revision history
hm	15 oct. 2007	rev 1.0
	original version

hm	19. oct 2007	rev 1.1
	manual mode was not detected because outputs were checked and not inputs UP and DN

hm	24. nov 2007	rev 1.2
	added shade_delay to avoid constant up and down if sun is out parcially

hm	8. feb 2009	rev 1.3
	added shading position shade_pos to be configured
	changed inputs to utilize calendar data structure

hm	13. mar. 2009	rev 1.4
	improved code

*)

END_FUNCTION_BLOCK

// POUs/Jalousie/BLIND_SHADE_S
FUNCTION_BLOCK BLIND_SHADE_S
VAR_INPUT
   UP, DN : BOOL;
   S_IN : BYTE;
   PI : BYTE;
   ENABLE : BOOL;
   SUN : BOOL;
   HORZ1 : REAL := 100.0;
   HORZ2 : REAL := 260.0;
   VERT : REAL := 90.0;
   ALERT: BOOL := FALSE;
END_VAR
VAR_IN_OUT
   CX : OSCAT_BASIC.calendar;
END_VAR
VAR_INPUT CONSTANT
   sunrise_offset : TIME := T#1h;
   sunset_preset : TIME := T#1h;
   shade_delay : TIME := T#60s;
   shade_pos : BYTE;
END_VAR
VAR_OUTPUT
   QU, QD : BOOL;
   STATUS : BYTE;
   PO : BYTE;
END_VAR
VAR
   sun_delay : OSCAT_BASIC.TOF;
END_VAR
(*
version 1.0	12. nov. 2009
programmer 	heinz
tested by		oscat


*)

(* status definition
   151 = shadow               move shutter down for shadowing
   152 = alert                  move shutter up by setting QU:=TRUE when door is open.
*)

(* the input sun is sent through tof which will delay the shade for the time shade_delay *)
sun_delay(IN := sun, PT := shade_delay);

IF ALERT THEN
   QU := TRUE;
   QD := FALSE;
   STATUS := 152;
ELSIF UP AND DN AND ENABLE AND sun_delay.Q
AND (CX.SUN_HOR > HORZ1) AND (CX.SUN_HOR < HORZ2)
AND (CX.SUN_VER < VERT)
AND (DT_TO_TOD(CX.UTC) > CX.SUN_RISE + sunrise_offset) AND (DT_TO_TOD(CX.UTC) < CX.SUN_SET - sunset_preset) THEN
   QU := UP;
   QD := DN;
   STATUS := 151;
   (* Calculate Position, must be shade_pos or less *)
   PO := MIN(PI, shade_pos);
ELSE
   QU := UP;
   QD := DN;
   PO := PI;
   STATUS := S_IN;
END_IF;



(* revision history
hf	12 nov. 2009	rev 1.0
	original version

*)

END_FUNCTION_BLOCK

// POUs/HLK/BOILER
FUNCTION_BLOCK BOILER
VAR_INPUT
	T_upper : REAL;
	T_lower : REAL;
	Pressure : BOOL := TRUE;
	enable : BOOL := TRUE;
	Req_1 : BOOL;
	Req_2 : BOOL;
	Boost : BOOL;
END_VAR
VAR_INPUT CONSTANT
	t_upper_min : REAL := 50.0;
	t_upper_max : REAL := 60.0;
	T_lower_enable : BOOL;
	T_lower_max : REAL := 60.0;
	T_request_1 : REAL := 70.0;
	T_request_2 : REAL := 50.0;
	T_request_hys : REAL := 5.0;
	T_protect_high : REAL := 80.0;
	T_protect_low : REAL := 10.0;
END_VAR
VAR_OUTPUT
	Heat : BOOL;
	error : BOOL;
	status : BYTE;
END_VAR
VAR
	edge: BOOL;
	boost_mode: BOOL;
	flag_0 : BOOL;
	flag_1: BOOL;
	flag_2: BOOL;
END_VAR

(*
version 1.2	13. mar. 2009
programmer 	hugo
tested by		oscat


this function block controls a hot water boiler. The Boiler can be equipped with two temperature sensors on top and bottom of the tank, T_LOWER_ENABLE must be set to True in this case.
alternatively can BOILER be configured for one (TOP) temperature sensor only (T_LOWER_ENABLE set to False).
A Pressure sensor is used to detect fresh water pressure and disable all heating if there is no water pressure. This input is dset to True by default, so if it is not used it can simply be left open.
A enable input enables the hot water heating while it is set to True. alternatively can a Ture on Req_1 or Req_2 start the heating to predefined temperatures during setup.
A low to high edge on the boost input will start heating imediately until T_upper_max is reached, it can be used to generate extra hot water when needed.

*)

(* read sensors and check for valid data *)
IF t_upper > t_protect_high THEN
	status := 1;
	heat := FALSE;
	error := TRUE;
ELSIF t_upper < t_protect_low THEN
	status := 2;
	heat :=	TRUE;
	error := TRUE;
ELSIF t_lower > T_protect_high AND t_lower_enable THEN
	status := 3;
	heat := FALSE;
	error := TRUE;
ELSIF t_lower < t_protect_low AND t_lower_enable THEN
	status := 4;
	heat := TRUE;
	error := TRUE;
ELSIF NOT pressure THEN
	status := 5;
	heat := FALSE;
	error := TRUE;
ELSIF req_1 OR req_2 OR enable OR boost THEN
	error := FALSE;

	(* determine if heat needs to be turned on *)
	IF boost AND NOT edge AND t_upper < t_upper_max THEN
		status := 101;
		heat := TRUE;
		boost_mode := TRUE;
	ELSIF enable AND t_upper < T_upper_min THEN
		status := 102;
		heat := TRUE;
	ELSIF req_1 AND t_upper < T_request_1 THEN
		status := 103;
		heat := TRUE;
	ELSIF req_2 AND t_upper < t_request_2 THEN
		status := 104;
		heat := TRUE;
	END_IF;

	(* determine the shut off temperature *)
	IF heat THEN
		IF (enable OR boost_mode) THEN
			flag_0 := TRUE;
			IF T_lower_enable AND T_lower > T_lower_max THEN
				flag_0 := boost_mode := FALSE;
			ELSIF NOT T_lower_enable AND T_upper > T_upper_max THEN
				flag_0 := boost_mode := FALSE;
			END_IF;
		ELSE
			flag_0 := FALSE;
		END_IF;
		flag_1 := (req_1 AND T_upper > T_request_1 + T_request_hys) AND req_1;
		flag_2 := (req_2 AND T_upper > T_request_2 + T_request_hys) AND req_2;

		(* shut off heat if no longer needed *)
		heat := flag_0 OR flag_1 OR flag_2;
		IF heat = FALSE THEN status := 100; END_IF;
	END_IF;
ELSE
	status := 100;
	heat := FALSE;
	error := FALSE;
END_IF;
edge := boost;


(* revision history
hm	27. feb. 2007	rev 1.0
	original version

hm	16. oct. 2008	rev 1.1
	improved performance

hm	13. mar. 2009	rev 1.2
	real constants updated to new systax using dot
	replaced double assignments
*)

END_FUNCTION_BLOCK

// POUs/Other/BUILDING_VERSION
FUNCTION BUILDING_VERSION : DWORD
VAR_INPUT
	IN : BOOL;
END_VAR


(*
version 1.1	16 dec 2007
programmer 	hugo
tested by		oscat

oscat_version returns the version number in dword format
132 is library version 1.32
if IN = true, the release date will be returned

*)

IF in THEN
	BUILDING_VERSION := DATE_TO_DWORD(D#2011-02-3);
ELSE
	BUILDING_VERSION := 100;
END_IF;

(* revision history
hm	6. oct 2006	rev 1.0
	original version

hm	16. dec 2007	rev 1.1
	added possibility to return date and version depending on IN.

*)

END_FUNCTION

// POUs/HLK/BURNER
FUNCTION_BLOCK BURNER
VAR_INPUT
	in : BOOL;
	stage2 : BOOL;
	over_temp : BOOL;
	oil_temp : BOOL := TRUE;
	Flame : BOOL;
	rst : BOOL;
	rst_timer : BOOL;
END_VAR
VAR_INPUT CONSTANT
	pre_heat_time : TIME := t#5s;
	pre_vent_time : TIME := t#15s;
	pre_ignite_time : TIME := t#5s;
	post_ignite_time : TIME := t#25s;
	stage2_delay : TIME := t#10s;
	safety_time : TIME := t#5s;
	lockout_time : TIME := t#10s;
	multiple_ignition : BOOL := TRUE;
	KW1 : REAL;
	KW2 : REAL;
END_VAR
VAR_OUTPUT
	motor : BOOL;
	coil1 : BOOL;
	coil2 : BOOL;
	pre_heat: BOOL;
	ignite : BOOL;
	KWh : REAL;
	status : BYTE;
	fail : BOOL;
END_VAR
VAR_IN_OUT
	runtime1 : UDINT;
	runtime2 : UDINT;
	cycles : UDINT;
END_VAR
VAR
	state : BYTE;
	last : TIME;
	tx: TIME;
	last_change: TIME;
	timer1 : OSCAT_BASIC.ONTIME;
	timer2 : OSCAT_BASIC.ONTIME;
	oil_temp_last: BOOL;
	cycles2 : UDINT;
END_VAR

(*
version 1.5	15 sep 2007
programmer 	oscat
tested by	oscat

burner ist eine Oel-Brenner_steuerung fuer nichtmodulierende Oelbrenner
die steuerung kann ueber setup werte programmiert werden und entsprechenden brennern angepasst werden.
die vorheizzeit ist die zeit die eine oelvorwaermung aufgeheizt wird bevor der motor gestartet wird.
der eingang oil_temp gibt an ob die oil_temp erreicht wurde, er ist default auf true und kann auch offen gelassen werden.
die vorbelueftungszeit ist die zeit die der luefter laeuft bevor die oelzufuhr freigegeben wird.
die vorzuendzeit iust diejenige zeit die die zuendung vor offnen des oelventiel gestartet wird.
nachzuendzeit ist die zeit die nach entzuendung der flamme noch gezuendet wird.
die sicherheitszeit ist die zeit nach der die oelzufuhr gesperrt wird wenn keine flamme entsteht.
nach ablauf der sicherheitszeit wird ein fehler flag gesetzt und kann erst nach der sperrzeit wieder durch einen reset geloescht werden.
waehrend der sperrzeit ist keine weitere zuendung oder einschalten moeglich.
das flag mehrfachzuendung gibt an ob eine erloschene flamme in betrieb automatisch wieder gezuendet werden soll.
der flammwaechster liegt auf eingang flamme, ein uebertemperaturschutz auf dem eingang over_temp
der betriebsstundenzaehler gibt die brennerstunden in stunden als real ausgabewer an.
der ausgang motor steuert den luefter / pumpenmotor, oil_ventil schaltet das oil ventil und zuendung schaltet die zuendung ein.

if output fail > 0 an error happened and the output has an error code:
0 :	no error
1 :	pre heating time expired and oil temp input is not true
2 :	flame monitor is active during preheating time
3 :	flame monitor active during pre_ventilation_time
4 :	no ignoition during safety time
5 :	no flame during operation
9 :	overtemp input is true

*)

(* read system time *)
tx := DWORD_TO_TIME(OSCAT_BASIC.T_PLC_MS());

(* check rst input and overtemp *)
IF rst OR over_temp OR state = 0 THEN
	IF status > 0 AND tx - last_change >= lockout_time AND rst THEN
		status := 110;
		fail := FALSE;
		state := 1;
	ELSE
		(* normaler reset *)
		motor := FALSE;
		coil1 := FALSE;
		coil2 := FALSE;
		ignite := FALSE;
		pre_heat := FALSE;
		IF over_temp THEN
			status := 9;
			fail := TRUE;
		END_IF;
		last_change := tx;
		last := tx;
		state := 1;
	END_IF;
END_IF;

(* check for timer rst and rst timer if true *)
IF rst_timer THEN
	runtime1 := 0;
	runtime2 := 0;
	cycles := 0;
	cycles2 := 0;
END_IF;

(* quit here if an error is present *)
IF (status > 0 AND status < 100) OR rst THEN RETURN; END_IF;

(* start sequence *)
CASE state OF

1:	(* in signal starts oil pre heating *)
	IF in AND flame THEN
		state := 7;
		pre_heat := FALSE;
		status := 2;
		last_change := tx;
	ELSIF in THEN
		pre_heat := TRUE;
		state := 2;
		last_change := tx;
	END_IF;

2:	(* after pre_heating time start motor *)
	IF (tx- last_change >= pre_heat_time AND oil_temp) OR (oil_temp AND NOT oil_temp_last) THEN
		motor := TRUE;
		state := 3;
		last_change := tx;
	(* pre_heat_time ist abgelaufen und oil_temp ist nicht aktiv *)
	ELSIF tx - last_change >= pre_heat_time AND NOT oil_temp THEN
		state := 7;
		pre_heat := FALSE;
		status := 1;
		last_change := tx;
	(* flame monitor cannot be active at this time *)
	ELSIF flame THEN
		state := 7;
		pre_heat := FALSE;
		status := 2;
		last_change := tx;
	END_IF;

3:	(* abwarten bis zündung eingeschaltet werden kann *)
	IF tx - last_change >= pre_vent_time - pre_ignite_time THEN
		ignite := TRUE;
		state := 4;
		last_change := tx;
	(* flame monitor cannot be active at this time *)
	ELSIF flame THEN
		state := 7;
		pre_heat := FALSE;
		motor := FALSE;
		status := 3;
		last_change := tx;
	END_IF;

4:	(* warten bis oelzufuhr geoeffnet werden darf *)
	IF tx - last_change >= pre_ignite_time THEN
		coil1 := TRUE;
		state := 5;
		last_change := tx;
	END_IF;

5:	(* warten auf flammwaechter und falls noetig abschalten *)
	IF tx - last_change >= safety_time OR flame THEN
		IF NOT flame THEN
			(* notabschaltung da flammwaechster nicht angesprochen hat *)
			state := 7;
			motor := FALSE;
			coil1 := FALSE;
			pre_heat := FALSE;
			ignite := FALSE;
			status := 4;
			last_change := tx;
		ELSE
			state := 6;
			last_change := tx;
		END_IF;
	END_IF;

6:	(* brenner läuft, flammueberwachung und nach ablauf der nachigniteszeit ignite abschalten *)
	IF NOT flame AND NOT multiple_ignition THEN
		(* notabschaltung da flammwaechster keine flamme meldet *)
		state := 7;
		motor := FALSE;
		coil1 := FALSE;
		coil2 := FALSE;
		pre_heat := FALSE;
		ignite := FALSE;
		status := 5;
		last_change := tx;
	ELSIF NOT flame AND multiple_ignition THEN
		ignite := TRUE;
		state := 5;
		coil2 := FALSE;
		last_change := tx;
	ELSE
		IF tx - last_change >= post_ignite_time THEN
			(* post_ignite_time abgelaufen, ignite abschalten *)
			ignite := FALSE;
		END_IF;
		IF tx - last_change >= stage2_delay AND stage2 THEN
			coil2 := TRUE;
		ELSE
			coil2 := FALSE;
		END_IF;
	END_IF;
END_CASE;

(* abschaltung wenn kein eingangssignal *)
IF NOT in THEN
	state := 1;
	motor := FALSE;
	coil1 := FALSE;
	coil2 := FALSE;
	ignite := FALSE;
	pre_heat := FALSE;
	last_change := tx;
END_IF;

(* runtimezähler *)
timer1(in := flame AND in AND motor AND coil1 AND NOT coil2, seconds := runtime1, cycles := cycles);
timer2(in := flame AND in AND motor AND coil1 AND coil2, seconds := runtime2, cycles := cycles2);
KWH := UDINT_TO_REAL(runtime1) * KW1 / 3600.0 + UDINT_TO_REAL(runtime2) * KW2 / 3600.0;

(* zeit fuer naechsten aufruf merken *)
last := tx;

(* set fail output IF ERROR and Status  if normal operation *)

IF status > 0 AND status < 100 THEN
	fail := TRUE;
ELSE
	fail := FALSE;
	IF NOT in THEN
		status := 110;
	ELSIF flame AND in AND motor AND coil2 AND coil1 THEN
		status := 113;
	ELSIF flame AND in AND motor AND coil1 THEN
		status := 112;
	ELSE
		status := 111;
	END_IF;
END_IF;



(*
31.12.2006	hm		rev 1.1
	added pre_heat timing and output
	flame monitor before ignition will generate error on status output
	added output for KWh

31.12.2006	hm		rev 1.2
	added oil_temp_input

31.12.2006	hm		rev 1.3
	changed status output to be byte instead of bool

22.1.2007		hm		rev 1.4
	renamed fail output to status
	added output cycles
	corrected an error while pre_heat would be on when an error was present
	added coil2 output and stage2 input

15.9.2007		hm		rev 1.5
	replaced Time() with T_PLC_MS for compatibility and performance reasons

hm	21. oct. 2008	rev 1.6
	changed code to use new ontime rev 2.0	
*)

END_FUNCTION_BLOCK

// POUs/HLK/DEW_RH
FUNCTION DEW_RH : REAL
VAR_INPUT
	VC : REAL;
	T : REAL;
END_VAR

(*
version 1.2	13. mar. 2009
programmer 	hugo
tested by		tobias

this function calculates the relative humidity in air for a given temperature in °C and vapor concentration in Kg/m³..

*)

DEW_RH := LIMIT(0.0, VC / DEW_CON(1.0, T), 100.0);

(* code before rev 1.1
dew_rh := VC / dew_con(100,T) * 100;
IF dew_rh > 100 THEN dew_rh := 100; END_IF;
*)

(* revision history
hm	29. apr 2007	rev 1.0
	original version

hm	2. 12. 2007	rev 1.1
	new code for better performance

hm	13. mar. 2009	rev 1.2
	real constants updated to new systax using dot

*)

END_FUNCTION

// POUs/HLK/DEW_TEMP
FUNCTION DEW_TEMP : REAL
VAR_INPUT
	RH : REAL;
	T : REAL;
END_VAR
VAR CONSTANT
	a : REAL := 7.5;
	b : REAL := 237.3;
END_VAR
VAR
	V : REAL;
END_VAR

(*
version 1.6	13. mar. 2009
programmer 	hugo
tested by		oscat

this function calculates the dew point for air given the temperature and relative humidity.
dew_temp(60,0.25) = 16.7 °C.
which means the dew point for air with 25° and 60% RH is at 16.7 °C.


*)

IF rh > 0.0 THEN
(*	old code was rewritten for better performance
	SDD := 6.1078*EXPT(10,(a*T)/(b+T));
	DD := RH/100 * SDD;
	V := LOG(DD/6.1078);
	dew_temp := b*V/(a-v);
*)
	V := LOG(RH * 0.01 * OSCAT_BASIC.EXP10((a*T) / (b+T)));
	DEW_TEMP := b*V / (a-V);
ELSE
	DEW_TEMP:= OSCAT_BASIC.phys.T0;
END_IF;

(* revision history

hm		2.10.2006	rev 1.0
	original version created

hm		29.4.2007	rev 1.1
	checked for rh not to be 0 because log(0) is not defined

hm		13.9.2007	rev 1.2
	code rewritten for better performance

hm	2. dec 2007	rev 1.3
	changed code for better performance

hm	8. jan 2008	rev 1.4
	further improvement in performance

hm	18. oct. 2008	rev 1.5
	using phys constants	

hm	13. mar. 2009	rev 1.6
	real constants updated to new systax using dot
	function will now return -273.15 °C for RH = 0
*)

(*
Bezeichnungen:
r = relative Luftfeuchte
T = Temperatur in °C
TK = Temperatur in Kelvin (TK = T + 273.15)
TD = Taupunkttemperatur in °C
DD = Dampfdruck in hPa
SDD = Sättigungsdampfdruck in hPa

Parameter:
a = 7.5, b = 237.3 für T >= 0
a = 7.6, b = 240.7 für T < 0 über Wasser (Taupunkt)
a = 9.5, b = 265.5 für T < 0 über Eis (Frostpunkt)

R* = 8314.3 J/(kmol*K) (universelle Gaskonstante)
mw = 18.016 kg (Molekulargewicht des Wasserdampfes)
AF = absolute Feuchte in g Wasserdampf pro m3 Luft

Formeln:

   1. SDD(T) = 6.1078 * 10^((a*T)/(b+T))
   2. DD(r,T) = r/100 * SDD(T)
   3. r(T,TD) = 100 * SDD(TD) / SDD(T)
   4. TD(r,T) = b*v/(a-v) mit v(r,T) = log10(DD(r,T)/6.1078)
   5. AF(r,TK) = 10^5 * mw/R* * DD(r,T)/TK; AF(TD,TK) = 10^5 * mw/R* * SDD(TD)/TK 

*)

END_FUNCTION

// POUs/electrical/DIMM_2
FUNCTION_BLOCK DIMM_2
VAR_INPUT
	SET : BOOL;
	VAL : BYTE := 255;
	I1 : BOOL;
	I2 : BOOL;
	RST : BOOL;
END_VAR
VAR_INPUT CONSTANT
	T_DEBOUNCE : TIME := T#10ms;
	T_ON_MAX : TIME := T#0h;
	T_DIMM_START : TIME := T#1s;
	T_DIMM: TIME := T#3s;
	MIN_ON : BYTE := 50;
	MAX_ON : BYTE := 255;
	RST_OUT : BOOL := TRUE;
	SOFT_DIMM : BOOL := TRUE;
	DBL1_TOG : BOOL;
	DBL2_TOG : BOOL;
	DBL1_SET : BOOL;
	DBL2_SET : BOOL;
	DBL1_POS : BYTE;
	DBL2_POS : BYTE;
END_VAR
VAR_OUTPUT
	Q : BOOL := FALSE;
	D1 : BOOL;
	D2 : BOOL;
END_VAR
VAR_IN_OUT
	OUT : BYTE;
END_VAR
VAR
	t1, t2 : OSCAT_BASIC.TOF;
	dc1, dc2 : CLICK_MODE;
	t3 : OSCAT_BASIC.TON;
	dim : OSCAT_BASIC._RMP_B;
END_VAR

(*
version 1.0	22. mar. 2009
programmer 	hugo
tested by	tobias

this is an intelligent dimmer interface with an autoset feature using double switch inputs
a configurable debounce timer will debounce the input signals
if t_on_max is set to anything other then 0 the output will be turned off after the max on time is reached.
the times for debounce, dimming ramp, wait time before dimming and max on time are all programmable.

the dimmer has outputs Q for on and off and also out with the analog dimm value.
two additional outputs d1 and d2 decode double clicks on i1 and i2.

*)

(* debouncing for inputs i1 and i2 *)
t1(IN := I1, PT := T_DEBOUNCE);
t2(IN := I2, PT := T_DEBOUNCE);
dc1(in := t1.Q, T_LONG := T_DIMM_START);
dc2(in := t2.Q, T_LONG := T_DIMM_START);


IF RST THEN
	IF RST_OUT THEN out := 0; END_IF;
	Q := FALSE;
	D1 := FALSE;
	D2 := FALSE;
ELSIF set THEN
	OUT := VAL;
	Q := TRUE;
ELSIF dc1.SINGLE THEN
	(* single click on i1 turns the dimmer on *)
	out := LIMIT(MAX(MIN_ON,1), out, MAX_ON);
	Q := TRUE;
ELSIF dc2.SINGLE THEN
	(* single click on i2 turns the dimmer off *)
	Q := FALSE;
ELSIF dc1.TP_LONG THEN
	(* continuous on at i1 dimms up *)
	IF NOT Q THEN
		out := SEL(SOFT_DIMM, LIMIT(MAX(MIN_ON,1), out, MAX_ON), 1);
	END_IF;
	Q := TRUE;
	dim.DIR := TRUE;
ELSIF dc2.TP_LONG THEN
	(* continuous on at i2 dimms down *)
	dim.DIR := FALSE;
END_IF;

(* set the double click output *)
IF NOT DBL1_TOG THEN D1 := FALSE; END_IF;
IF dc1.DOUBLE THEN
	IF DBL1_SET THEN
		OUT := DBL1_POS;
		Q := TRUE;
	ELSE
		D1 := NOT D1;
	END_IF;
END_IF;
IF NOT DBL2_TOG THEN D2 := FALSE; END_IF;
IF dc2.DOUBLE THEN
	IF DBL2_SET THEN
		OUT := DBL2_POS;
		Q := TRUE;
	ELSE
		D2 := NOT D2;
	END_IF;
END_IF;


(* while dimming is active ramp the output out up or down *)
dim(dir := dc2.LONG, e := dc1.LONG OR dc2.LONG , TR := T_DIMM, rmp := out);

(* turn off output if a value of 0 is reached *)
IF out = 0 THEN Q := FALSE; END_IF;

(* limit the maximum runtime *)
IF t_ON_MAX > t#0s THEN
	t3(in := q, pt := T_ON_MAX);
	Q := Q XOR t3.Q;
END_IF;




(* revision history

hm 22. mar. 2009	rev 1.0
	original version

*)

END_FUNCTION_BLOCK

// POUs/electrical/DIMM_I
FUNCTION_BLOCK DIMM_I
VAR_INPUT
	SET : BOOL;
	VAL : BYTE := 255;
	IN : BOOL;
	RST : BOOL;
END_VAR
VAR_INPUT CONSTANT
	T_DEBOUNCE : TIME := T#10ms;
	T_RECONFIG : TIME := T#10s;
	T_ON_MAX : TIME := T#0h;
	T_DIMM_START : TIME := T#1s;
	T_DIMM: TIME := T#3s;
	MIN_ON : BYTE := 50;
	MAX_ON : BYTE := 255;
	SOFT_DIMM : BOOL := TRUE;
	DBL_toggle : BOOL;
	RST_OUT : BOOL;
END_VAR
VAR_OUTPUT
	Q : BOOL := FALSE;
	DBL : BOOL;
END_VAR
VAR_IN_OUT
	OUT : BYTE;
END_VAR
VAR
	config : SW_RECONFIG;
	decode : CLICK_MODE;
	t3 : OSCAT_BASIC.TON;
	dim : OSCAT_BASIC._RMP_B;
	dir : BOOL;
END_VAR

(*
version 2.3	26. jan. 2009
programmer 	hugo
tested by		tobias

this is an intelligent dimmer interface with an autoset feature for "in" it will automatically detect the type of switch:
low active pulses or high high active pulses are allowd for in.
a configurable debounce timer will debounce input signals
if t_on_max is set to anything other then 0 the output will be turned off after the max on time is reached.
the times for debounce, dimming ramp, wait time before dimming and max on time are all programmable.

the dimmer has outputs Q for on and off and also out with the analog dimm value.

*)

(* the input is first sent through auto reconfiguration and debouncing *)
config(IN := IN, TD := T_DEBOUNCE, TR := T_RECONFIG);
decode(in := config.Q, T_LONG := T_DIMM_START);

IF RST THEN
	IF rst_out THEN out := 0; END_IF;
	Q := FALSE;
	dir := out > 127;
ELSIF set THEN
	out := val;
	Q := TRUE;
	(* set direction to up when value < 127 otherwise set dir down dir is reversed because next action will reverse again *)
	dir := out > 127;
ELSIF decode.SINGLE THEN
	(* a single click reverses output Q *)
	Q := NOT Q;
	(* when dimmer is turned on we need to limit out to min and max limits *)
	IF Q THEN	out := LIMIT(MAX(MIN_ON,1), out, MAX_ON);	END_IF;
	(* set the appropriate direction of dimmer dir is reversed because next action will reverse again *)
	dir := out > 127;
ELSIF decode.TP_LONG THEN
	IF NOT Q THEN
		IF SOFT_DIMM THEN
			OUT := 1;
			dir := TRUE;
		ELSE
			OUT := LIMIT(MAX(MIN_ON,1), out, MAX_ON);
			DIR := out < 127;
		END_IF;
		Q := TRUE;
	ELSE
		(* reverse direction with every long click *)
		dir := NOT dir;
	END_IF;
END_IF;

(* set the double click output *)
IF NOT dbl_toggle THEN dbl := FALSE; END_IF;
IF decode.DOUBLE THEN dbl := NOT dbl; END_IF;

(* while dimming is active ramp the output out up or down *)
dim(DIR := dir, e := decode.LONG AND Q, TR := T_DIMM, rmp := out);

(* reverse direction when limits are reached *)
IF out = 0 THEN
	dir := TRUE;
ELSIF out = 255 THEN
	dir := FALSE;
END_IF;

(* limit the maximum runtime *)
IF t_ON_MAX > t#0s THEN
	t3(in := q, pt := T_ON_MAX);
	Q := Q XOR t3.Q;
END_IF;




(* revision history

hm 22.1.2007		rev 1.1
	deleted unused structure ramp

hm 2.feb 2007		rev 1.2
	changed structure to read time() at the beginning for better time consistency if a higher priorized tak interrupts dimm_i
	added statements in case structure for state 1 to allow for short 1 cycle input pulses

hm 	15.9.2007		rev 1.3
	replaced Time() with T_PLC_MS for compatibility and performance reasons

hm	30. sep. 2008	rev 1.4
	added Input VAL to supply value for set input
	added setup parameter init_val

hm	22. oct. 2008	rev 2.0
	new code and features

hm	14. nov. 2008	rev 2.1
	added soft_dimm feature

hm	16. nov. 2008	rev 2.2
	added reset out feature

hm	26. jan. 2009	rev 2.3
	dimming will also reverse at out = 0
	rst will override set
*)

END_FUNCTION_BLOCK

// POUs/electrical/F_LAMP
FUNCTION_BLOCK F_LAMP
VAR_INPUT
	SWITCH : BOOL;
	DIMM : BYTE := 255;
	RST : BOOL;
END_VAR
VAR_OUTPUT
	LAMP : BYTE;
	STATUS : BYTE;
END_VAR
VAR_IN_OUT
	ONTIME : UDINT;
	CYCLES : UDINT;
END_VAR
VAR_INPUT CONSTANT
	T_NO_DIMM : UINT := 100;
	T_MAINTENANCE : UINT := 15000;
END_VAR
VAR
	runtime : OSCAT_BASIC.ONTIME;
END_VAR

(*
version 1.2	22. oct. 2008
programmer 	hugo
tested by	oscat

F_Lamp is an interface to flourescent lamps. its main purpose is to protect flourescent lamps from dimming within the first T_NO_DIMM Time.
If Flourescent Lamps are dimmed during the first 100 hours the lifetime of the lamp is reduced dramatically.
The interface also counts ontime and cycles of the lamp for maintanance purposes.

*)

runtime(in := switch, seconds := ontime, cycles := cycles);

IF RST THEN
	ONTIME := 0;
	CYCLES := 0;
END_IF;
IF SWITCH THEN
	IF ontime < T_NO_DIMM * 3600 THEN
		LAMP := 255;
		STATUS := 111;
	ELSE
		LAMP := DIMM;
		STATUS := 112;
	END_IF;
ELSE
	LAMP := 0;
	STATUS := 110;
END_IF;


IF ontime >= T_maintenance * 3600 AND T_Maintenance > 0 THEN
	status := 120;
END_IF;



(* revision history
hm	8. feb. 2007	rev 1.1
	original version

hm	22. oct. 2008	rev 1.2
	changed use of ontime for ontime 2.0
	ontime is now in seconds not hours
*)

END_FUNCTION_BLOCK

// POUs/HLK/HEAT_INDEX
FUNCTION HEAT_INDEX : REAL
VAR_INPUT
	T : REAL;
	RH : REAL;
END_VAR
VAR
	RH2 : REAL;
	T2 : REAL;
END_VAR

(*
version 1.3	13. mar. 2009
programmer 	hugo
tested by		tobias

this function calculates the heat index temperature depending on external temperature and Relative humidity

*)

IF RH < 20.0 OR T < 20.0 THEN
	HEAT_INDEX := T;
ELSE
	RH2 := RH * RH;
	T := OSCAT_BASIC.C_TO_F(T);
	T2 := T * T;
	HEAT_INDEX := -42.379 + 2.04901523 * T - 6.83783E-3 * T2
			+ RH * (10.1433127 - 0.22475541 * T + 1.22874E-3 * T2)
			+ RH2 * (8.5282E-4 * T - 5.481717E-2 - 1.99E-6 * T2);
	HEAT_INDEX := OSCAT_BASIC.F_TO_C(HEAT_INDEX);
END_IF;

(* revision history

hm 27.2.2007		rev 1.1
	deleted unused variables rh3 and T3

hm	2.12.2007		rev 1.2
	changed code for better performance

hm	13. mar. 2009	rev 1.3
	real constants updated to new systax using dot

*)

END_FUNCTION

// POUs/HLK/HEAT_METER
FUNCTION_BLOCK HEAT_METER
VAR_INPUT
	TF, TR : REAL;
	LPH : REAL;
	E : BOOL;
	RST : BOOL;
END_VAR
VAR_INPUT CONSTANT
	CP : REAL;
	Density : REAL;
	Content : REAL;
	Pulse_Mode : BOOL;
	Return_meter : BOOL;
	AVG_time : TIME := T#5s;
END_VAR
VAR_OUTPUT
	C : REAL;
END_VAR
VAR_IN_OUT
	Y : REAL;
END_VAR
VAR
	tx, last : DWORD;
	int1 : OSCAT_BASIC.FT_INT2;
	edge : BOOL;
	x: REAL;
	init: BOOL;
	y_last: REAL;
END_VAR

(*
version 1.10	23. jan. 2011
programmer 		hugo
tested by		oscat

Heat meter measures the heat transfer of water of a mixture of water and another component.
The inputs are foreward temperature and reverse temperature.
the additional component is specified with its parameters density, Specific heat capacity and content in %.
an input e anables the measurement while it can be configured to be based on X liters / pulse or in liters / hour.
the output Y is in Joule.

*)

IF rst THEN
	int1(rst := TRUE);
	int1.rst := FALSE;
	C := 0.0;
	Y := 0.0;
ELSIF e THEN
	X := (WATER_DENSITY(SEL(return_meter, TF, TR), FALSE) * (WATER_ENTHALPY(TF) - WATER_ENTHALPY(TR)) * (1.0 - content) + CP * Density * content * (TF-TR));
END_IF;

(* integrate or add consumption *)
int1(run := NOT pulse_mode AND e, in := X * LPH * 2.77777777777E-4);
IF pulse_mode THEN
	IF NOT edge AND E THEN Y := Y + X * LPH; END_IF;
ELSE
	Y := int1.Out;
END_IF;

(* store the value of e *)
edge := e;

(* read system_time *)
tx := OSCAT_BASIC.T_PLC_MS();

(* only init at startup necessary *)
IF NOT init THEN
	init := TRUE;
	last := tx;
END_IF;

(* calculate the current consumption *)
IF (tx - last >= TIME_TO_DWORD(AVG_TIME)) AND (avg_time > T#0s) THEN
	last := tx;
	C := (Y - Y_last) * 3.6E6 / DWORD_TO_REAL(TIME_TO_DWORD(AVG_TIME));
	Y_last := Y;
END_IF;



(* revision history
hm	16. nov. 2007	rev 1.0
	original version

hm	24. dec. 2007	rev 1.1
	added config variable return_meter
	added output C for current consumption

hm	6. mar. 2008	rev 1.2
	corrected an error in pulse mode

hm	16. mar. 2008	rev 1.3
	added type conversion to avoid warnings under codesys 3.0

hm	21. oct. 2008	rev 1.4
	improved code

hm	6. nov. 2008	rev 1.5
	changed to FT_INT2 to avoid overrun at hig values

hm	8. feb. 2009	rev 1.6
	changes Y to be I/O

hm	23. mar. 2009	rev 1.7
	real constants updated to new systax using dot
	corected error in formula

hm	27. jul 2009	rev 1.8
	output C is now calculated in J/h

hm	13. nov. 2009	rev 1.9
	output C is now calculated correctly

hm	23. jan. 2011	rev 1.10
	corrected an error with pulse_mode
*)

END_FUNCTION_BLOCK

// POUs/HLK/WATER_DENSITY
FUNCTION WATER_DENSITY : REAL
VAR_INPUT
	T : REAL;
	Sat : BOOL;
END_VAR
VAR CONSTANT
	a0 : REAL := 999.83952;
	a1 : REAL := 16.952577;
	a2 : REAL := -7.9905127E-3;
	a3 : REAL := -4.6241757E-5;
	a4 : REAL := 1.0584601E-7;
	a5 : REAL := -2.8103006E-10;
	b  : REAL := 0.0168872;
END_VAR
VAR
	T2: REAL;
	T4: REAL;
END_VAR


(*
version 1.2	13. mar. 2009
programmer 	hugo
tested by		tobias

this function calculates the water density for air free water between 0 and 100 deg C
while sat is false the denisty is calculated for air free water and when sat = true
the calculation is performed for water saturated with air.

*)

T2 := T * T;
T4 := T2 * T2;
WATER_DENSITY := (a0 + a1*T + a2*T2 + a3*T2*T + a4*T4 + a5*T4*T) / (1.0 + b*T);
IF sat THEN WATER_DENSITY := WATER_DENSITY - 0.004612 + 0.000106 * T; END_IF;


(* revision history

hm	13.9.2007		rev 1.0
	original version

hm	2.12.2007		rev 1.1
	changed code for better performance

hm	13. mar. 2009	rev 1.2
	real constants updated to new systax using dot

*)

(*
    °C - die Celsius-Temperatur in Grad Celsius
    v – das spezifische Volumen in Kubikdezimeter je Kilogramm dm³/kg
    h – die spezifische Enthalpie in Kilojoule je Kilogramm 	kJ/kg
    u – die spezifische Innere Energie in Kilojoule je Kilogramm 	kJ/kg
    s – die spezifische Entropie in Kilojoule je Kilogramm mal Kelvin 	kJ/(kg·K)
    cp - die spezifische Wärmekapazität bei konstantem Druck in Kilojoule je Kilogramm mal Kelvin 	kJ/(kg·K)
    Y – Volumenausdehnungskoeffizient in 10-3 durch Kelvin  10-3/K
    L – Wärmeleitfähigkeit in Milliwatt je Meter mal Kelvin  mW / (m·K) 
    n – Viskosität in Mikropascal mal Sekunde uPa·s 	
    s ? – Oberflächenspannung in Millinewton je Meter  mN/m


°C 		v 				h 			u 		s 			cp 		Y 		L		n		s	
-20		1,006580	
0 		1,000160 		0,06 		-0,04 	-0,0001 	4,228 	-0,080 	561,0 	1792 	75,65
4		1,000028
5 		1,0000 		21,1 		21,0 	0,076 		4,200 	0,011 	570,6 	1518 	74,95
10 		1,0003 		42,1 		42,0 	0,151 		4,188 	0,087 	580,0 	1306 	74,22
15 		1,0009 		63,0 		62,9 	0,224 		4,184 	0,152 	589,4 	1137 	73,49
20 		1,001797 		83,9 		83,8 	0,296 		4,183 	0,209 	598,4 	1001 	72,74
25 		1,0029 		104,8 		104,7 	0,367 		4,183 	0,259 	607,2 	890,4 	71,98
30 		1,0044 		125,8 		125,7 	0,437 		4,183 	0,305 	615,5 	797,7 	71,20
35 		1,0060 		146,7 		146,6 	0,505 		4,183 	0,347 	623,3 	719,6 	70,41
40 		1,007842 		167,58 	167,5 	0,572 		4,182 	0,386 	630,6 	653,3 	69,60
45 		1,0099 		188,5 		188,4 	0,638 		4,182 	0,423 	637,3 	596,3 	68,78
50 		1,0121 		209,4 		209,3 	0,704 		4,181 	0,457 	643,6 	547,1 	67,95
60 		1,017089 		251,2 		251,1 	0,831 		4,183 	0,522 	654,4 	466,6 	66,24
70 		1,0227 		293,1 		293,0 	0,955 		4,187 	0,583 	663,1 	404,1 	64,49
80 		1,029027 		335,0 		334,9 	1,075 		4,194 	0,640 	670,0 	354,5 	62,68
90 		1,0359 		377,0 		376,9 	1,193 		4,204 	0,696 	675,3 	314,6 	60,82
99,63 	1,0431 		417,5 		417,4 	1,303 		4,217 	0,748 	679,0 	283,0 	58,99
100	1,043453		419,1

Stoffdaten von Wasser Quelle Wickipedia

*)

END_FUNCTION

// POUs/HLK/WATER_ENTHALPY
FUNCTION WATER_ENTHALPY : REAL
VAR_INPUT
	T : REAL;
END_VAR
VAR
	Pts : INT := 11;
	data : ARRAY[1..20, 0..1] OF REAL := [0.0,0.06, 10.0,42.1, 20.0,83.9, 30.0,125.8, 40.0,167.58, 50.0,209.4, 60.0,251.2, 70.0,293.1, 80.0,335.0, 90.0,377.0, 100.0,419.1];
END_VAR

(*
version 1.1	13. mar. 2009
programmer 	hugo
tested by		tobias

water_enthalpy calculates the enthalpy of liquid water from 0..100 °C 

*)

WATER_ENTHALPY := OSCAT_BASIC.LINEAR_INT(T, Data, Pts);



(*
    °C - die Celsius-Temperatur in Grad Celsius
    v – das spezifische Volumen in Kubikdezimeter je Kilogramm dm³/kg
    h – die spezifische Enthalpie in Kilojoule je Kilogramm 	kJ/kg
    u – die spezifische Innere Energie in Kilojoule je Kilogramm 	kJ/kg
    s – die spezifische Entropie in Kilojoule je Kilogramm mal Kelvin 	kJ/(kg·K)
    cp - die spezifische Wärmekapazität bei konstantem Druck in Kilojoule je Kilogramm mal Kelvin 	kJ/(kg·K)
    Y – Volumenausdehnungskoeffizient in 10-3 durch Kelvin  10-3/K
    L – Wärmeleitfähigkeit in Milliwatt je Meter mal Kelvin  mW / (m·K) 
    n – Viskosität in Mikropascal mal Sekunde uPa·s 	
    s ? – Oberflächenspannung in Millinewton je Meter  mN/m


°C 		v 				h 			u 		s 			cp 		Y 		L		n		s	
-20		1,006580	
0 		1,000160 		0,06 		-0,04 	-0,0001 	4,228 	-0,080 	561,0 	1792 	75,65
4		1,000028
5 		1,0000 		21,1 		21,0 	0,076 		4,200 	0,011 	570,6 	1518 	74,95
10 		1,0003 		42,1 		42,0 	0,151 		4,188 	0,087 	580,0 	1306 	74,22
15 		1,0009 		63,0 		62,9 	0,224 		4,184 	0,152 	589,4 	1137 	73,49
20 		1,001797 		83,9 		83,8 	0,296 		4,183 	0,209 	598,4 	1001 	72,74
25 		1,0029 		104,8 		104,7 	0,367 		4,183 	0,259 	607,2 	890,4 	71,98
30 		1,0044 		125,8 		125,7 	0,437 		4,183 	0,305 	615,5 	797,7 	71,20
35 		1,0060 		146,7 		146,6 	0,505 		4,183 	0,347 	623,3 	719,6 	70,41
40 		1,007842 		167,58 	167,5 	0,572 		4,182 	0,386 	630,6 	653,3 	69,60
45 		1,0099 		188,5 		188,4 	0,638 		4,182 	0,423 	637,3 	596,3 	68,78
50 		1,0121 		209,4 		209,3 	0,704 		4,181 	0,457 	643,6 	547,1 	67,95
60 		1,017089 		251,2 		251,1 	0,831 		4,183 	0,522 	654,4 	466,6 	66,24
70 		1,0227 		293,1 		293,0 	0,955 		4,187 	0,583 	663,1 	404,1 	64,49
80 		1,029027 		335,0 		334,9 	1,075 		4,194 	0,640 	670,0 	354,5 	62,68
90 		1,0359 		377,0 		376,9 	1,193 		4,204 	0,696 	675,3 	314,6 	60,82
99,63 	1,0431 		417,5 		417,4 	1,303 		4,217 	0,748 	679,0 	283,0 	58,99
100	1,043453		419,1

Stoffdaten von Wasser Quelle Wickipedia

Wasser hat unter Normaldruck seine größte Dichte von 1000 Kilogramm pro Kubikmeter bei 3,98 °C und zeigt damit eine Dichteanomalie. 
Diese besteht darin, dass sich Wasser unterhalb von 3,98 °C bei weiterer Temperaturverringerung, auch beim Wechsel zum festen 
Aggregatzustand, wieder ausdehnt, was man nur von wenigen Stoffen kennt. Die derzeit genauesten publizierten Werte für die maximale 
Dichte liegen bei (999,974950 ± 0,00084) kg/m³ und bei (3,983 ± 0,00067) °C für die Temperatur, bei der dieser Wert erreicht wird. 
Die Werte stellen einen Mittelwert der von verschiedenen physikalischen Instituten veröffentlichten Zahlen dar (Stand 2001).

Die Berechnung der Dichte von luftfreiem Wasser DLF in Abhängigkeit von der Temperatur T ([T] = °C) kann mit Hilfe der folgenden 
Virialgleichung erfolgen:
: \frac{D_{\rm LF}}{\rm g/l} = \frac{a_0 + a_1 T + a_2 T^2 + a_3 T^3 + a_4 T^4 + a_5 T^5}{1 + b T}.
mit den Koeffizienten: a0 = 999,83952; a1 = 16,952577 (°C)-1; a2 = -7,9905127·10-3 (°C)-2; a3 = -4,6241757·10-5 (°C)-3; 
a4 = 1,0584601·10-7 (°C)-4; a5 = -2,8103006·10-10 (°C)-5 und b = 0,0168872. 
Für die Berechnung der Dichte von luftgesättigtem Wasser korrigiert man den Wert nach 
DLG/(g/l) = DLF/(g/l) - 0,004612 + 0,000106 (°C)-1·T. (Quelle: PTB-Mitteilungen 100/3-90)

*)

(* revision history
hm	13. mar. 2009	rev 1.0
	original version

hm	13. mar. 2009	rev 1.1
	real constants updated to new systax using dot

*)

END_FUNCTION

// POUs/HLK/HEAT_TEMP
FUNCTION_BLOCK HEAT_TEMP
VAR_INPUT
	T_EXT : REAL;
	T_INT : REAL;
	OFFSET : REAL;
	T_REQ : REAL;
END_VAR
VAR_INPUT CONSTANT
	TY_MAX : REAL := 70.0;
	TY_MIN : REAL := 25.0;
	TY_CONFIG : REAL := 70.0;
	T_INT_CONFIG : REAL := 20.0;
	T_EXT_CONFIG : REAL := -15.0;
	T_DIFF : REAL := 10.0;
	C : REAL := 1.33;
	H : REAL := 3.0;
END_VAR
VAR_OUTPUT
	TY : REAL;
	HEAT : BOOL;
END_VAR
VAR
	tr : REAL;
	tx: REAL;
END_VAR

(*
version 1.2	13. mar. 2009
programmer 	hugo
tested by		oscat

Heat_Temp calculates a heat characteristic based on the formula: tv=ti+(tvmax-ti)*((ti-tau)/(ti-taumin))^(1/n)
while
tv necessary heating temperature.
ti internal room temperature (20°C)
tau current external temperature
taumin external temperature to determine characteristics
C exponent for heating system (normally 1,33 or 1,1 for floor heating)

The two additional inputs TY_min and TY_max set limits for the output TY, while an offset inputs allows to rise or lower the room temperature.

*)

tr := T_INT + OFFSET;
tx := (tr - T_EXT) / (T_INT_CONFIG - T_EXT_CONFIG);

IF T_EXT + H > tr THEN
	TY := 0.0;
ELSE
	TY := LIMIT(TY_MIN, tr + T_DIFF * 0.5 * tx + (TY_CONFIG - T_DIFF * 0.5 - tr) * EXPT(tx, 1.0 / C), TY_MAX);
END_IF;

TY := MAX(TY, T_REQ);
HEAT := TY > 0.0;


(*

tv=ti+(tvmax-ti)*((ti-tau)/(ti-taumin))^(1/n)

tv aktuelle Vorlauftemp.
ti Raumtemperatur innen (20°C)
tau aktuelle Außentemperatur
taumin minimale Außentemperatur -12°C oder -15°C
n Heizkörperexponent (meistens 1,33)
Fußbodenheizung = 1,1
Wandheizung 1,3

Normen z. B. DIN 4703, DIN 4725 oder die Literatur, z. B Recknagel Abschnitt 1.3.5.

*)


(* revision history
hm	27. jan. 2008	rev 1.0
	original version

hm	26. sep. 2008	rev 1.1
	moved T_INT from config to Input
	added config variable H
	corrected error in formula

hm	13. mar. 2009	rev 1.2
	improved code

*)

END_FUNCTION_BLOCK

// POUs/HLK/LEGIONELLA
FUNCTION_BLOCK LEGIONELLA
VAR_INPUT
	manual : BOOL;
	temp_boiler : REAL;
	temp_return : REAL := 100.0;
	DT_in: DT;
	rst : BOOL;
END_VAR
VAR_INPUT CONSTANT
	T_start: TOD := tod#03:00:00;
	day : INT := 7;
	temp_set : REAL := 70.0;
	temp_offset : REAL := 10.0;
	temp_hys : REAL := 5.0;
	t_max_heat: TIME := t#10m;
	t_max_ret : TIME := t#10m;
	tp_0: TIME := t#5m;
	TP_1: TIME := t#5m;
	tp_2: TIME := t#5m;
	tp_3: TIME := t#5m;
	tp_4: TIME := t#5m;
	tp_5: TIME := t#5m;
	tp_6: TIME := t#5m;
	tp_7: TIME := t#5m;
END_VAR
VAR_OUTPUT
	Heat : BOOL;
	pump : BOOL;
	valve0 : BOOL;
	valve1 : BOOL;
	valve2 : BOOL;
	valve3 : BOOL;
	valve4 : BOOL;
	valve5 : BOOL;
	valve6 : BOOL;
	valve7 : BOOL;
	run: BOOL;
	Status : BYTE;
END_VAR
VAR
	X1: TIMER_1;
	x2: OSCAT_BASIC.SEQUENCE_8;
	x3: OSCAT_BASIC.HYST_1;
	init: BOOL;
END_VAR

(*
version 1.3	13. mar. 2009
programmer 	oscat
tested by		oscat

Legionella is a complete sequencer for up to 8 hot water lines that need to be sterilzed periodically.
legionella needs a DT input with the appropriate time, usually gererated by the rtc of the system. for system independence this time is connected externally.
T_start is the time when sterilazation should be started and day is the day_of_week when it should be performed (1=Monday and 7=sunday).
so sterilazation is autioimatically performed once a week at a specified time.
temp_set and temp_hys and temp_offset specify the boiler temperatur nedded for sterilization. as a defaut Temp_set is set to 70 deg C and Temp_hys is set to 5 deg C and temp_offset is 10 deg C.
a temp boiler input reads the boiler temperature of the hot water tank.
after a start pulse is gererated by the weekly timer or a manual test input the sequence is started:
1. the boiler is heated to temp_set + temp_offset + temp_hys = 85 deg C unless chaged at setup.
	the heat output is turned on and tells the heater to turn heating on. if the temp is not reached for a time of t_max_heat (10 min) the error output is set and the sequence is stopped.
2. after the specified temperature is reached, the output valve0 and pump is turned on and starts sterilization of line0 until temp_return has reached temp_set and continues to sterilize for a time of tp_0 (5 min default).
	if tmep_set is not reached at the temp_return_input then the error output is set and the sequence will be stopped.
	if there is no temp sensor for temp_return (the temperature at the return point for the circulation pump pls set this imput to a value greater then temp_set (by default use 100 deg C).
	in this case sterilization is performed for the default times without monitoring the return temp.
3. this sequence is repeated for up to valves.

connection scheme:

temp_boiler:	input oif the boiler temperature sensor.
temp_hys:		config value for the heater hysteresis, preset to 5 deg C.
temp_offset:	config value for the heater temp_offset against temp_set, preset to 10 deg C.
temp_set:		config value for the specified sterilization temperature, preset to 70 deg C.
temp_return:	input of the circulation return line temperature sensor, if not availabe set this value to 100 deg C.
manual:		manual input to start the sterilization by hand for diagnostic purposes, rising edge active, leave low for automatic operation.
DT_in:			date,time input supplied by a external real time clock.
T_start:		time of day when the sterilization should be started.
day:			config value for day of week when the process should be started, preset to sunday.
t_max_hest:	tmax time to be needed for the heater to heat the hot water tank to the specified value, preset to 10 min.

*)

(* startup initialization *)
IF NOT init THEN
	init := TRUE;
	X1.day := SHR(BYTE#128,day);
	X1.start := T_start;
	X3.low := Temp_offset + temp_set;
	X3.high := Temp_hys + X3.low;
	X2.wait0 := T_max_heat;
	X2.delay0 := TP_0;
	X2.delay1 := TP_1;
	X2.delay2 := TP_2;
	X2.delay3 := TP_3;
	X2.delay4 := TP_4;
	X2.delay5 := TP_5;
	X2.delay6 := TP_6;
	X2.delay7 := TP_7;
	X2.wait1 := T_max_ret;
	X2.wait2 := T_max_ret;
	X2.wait3 := T_max_ret;
	X2.wait4 := T_max_ret;
	X2.wait5 := T_max_ret;
	X2.wait6 := T_max_ret;
	X2.wait7 := T_max_ret;
	X2();
END_IF;

(* oerational code *)
X1(DTi := DT_in);
IF X1.Q OR MANUAL OR x2.run THEN
	X3(in := temp_boiler);
	X2.in0 := X3.Q OR x3.win;
	X2.in1 := temp_return >= temp_set;
	X2.in2 := x2.in1;
	X2.in3 := x2.in1;
	X2.in4 := x2.in1;
	X2.in5 := x2.in1;
	X2.in6 := x2.in1;
	X2.in7 := x2.in1;
	X2.rst := rst;
	X2(start := X1.Q OR MANUAL);
	run := x2.run;
	pump := x2.qx;
	Heat := NOT X3.Q AND x2.run;
	valve0 := X2.Q0;
	valve1 := X2.Q1;
	valve2 := X2.Q2;
	valve3 := X2.Q3;
	valve4 := X2.Q4;
	valve5 := X2.Q5;
	valve6 := X2.Q6;
	valve7 := X2.Q7;
	pump := X2.qx;
	status := X2.status;
ELSE;
	X2(start :=0);
	status := x2.status;
END_IF;

(* revision history

hm 17.jan 2007	rev 1.1
	rewritten to st for higher performance
	changes eeror output to esr compatible status output

hm	23. 10.2008	rev 1.2
	update code to use new version of timer_1

hm	13. mar. 2009	rev 1.3
	real constants updated to new systax using dot
	using new module sequence_8
*)

END_FUNCTION_BLOCK

// POUs/electrical/TIMER_1
FUNCTION_BLOCK TIMER_1
VAR_INPUT
	E : BOOL := TRUE;
	DTI : DT;
	START : TOD;
	DURATION : TIME;
	DAY : BYTE := 2#0111_1111;
END_VAR
VAR_OUTPUT
	Q : BOOL;
	stop : TIME;
END_VAR


(*
version 2.2	16. dec. 2009
programmer 	oscat
tested by		oscat

this is a simple timer that generates an output pulse on selected days.
the output pulse width can be programmed with duration, if set to 0 no pulse is generated.
day specifies the specific days for the event to occur, bit 0 = sunday, bit 1 = saturday, bit 2 = friday ....
for all days to be active 127 has to be specified for DAY.

*)

IF E THEN
	stop := TOD_TO_TIME(START) + DURATION;
	IF stop > T#24h THEN stop := stop - T#24h; END_IF;
	Q := OSCAT_BASIC.TIMECHECK(DT_TO_TOD(DTI), START, TIME_TO_TOD(stop)) AND (SHR(BYTE#128, OSCAT_BASIC.DAY_OF_WEEK(DT_TO_DATE(DTI))) AND DAY) > BYTE#0;
ELSE
	Q := FALSE; (* clear output when e is not true *)
END_IF;


(*
1.12.2006 hm		rev 1.1
	corrected an error with pulse width = 0.

25.12.2006 hm		rev 1.2
	corrected an error when timer overflows.

14.apr 2007 hm		rev 1.3
	corrected an error while while output would not go active when start year would be 1970.
	increase accuracy by checking every 100ms
	added init section to compensate for timer overflow

15.9.2007 hm		rev 1.4
	replaced Time() with T_PLC_MS for compatibility and performance reasons

hm	1. okt 2007		rev 1.5
	corrected an error while output would not stay active over midnight.

hm	17. jan 2008	rev 1.6
	New code with better performance  
	Output is now only active during the time of day it is supposed to 
	no pulse is generated at power up

hm	7. oct. 2008	rev 1.7
	changed function weekday to day_of_week

hm	23. oct. 2008	rev 2.0
	new code, added input E, now days can be selected by bits in byte day

hm	6. nov. 2008	rev 2.1
	added default for input EN and input DAY

hm 16. dec 2009	rev 2.2
	fixed a bug over midnight

*)

END_FUNCTION_BLOCK

// POUs/electrical/PULSE_LENGTH
FUNCTION_BLOCK PULSE_LENGTH
VAR_INPUT
	in : BOOL;
END_VAR
VAR_OUTPUT
	short : BOOL;
	middle : BOOL;
	long : BOOL;
END_VAR
VAR_INPUT CONSTANT
	T_short : TIME := t#100ms;
	T_long : TIME := t#1s;
END_VAR
VAR
	tx : TIME;
	tn: TIME;
	edge : BOOL;
END_VAR

(*
version 1.1	15 sep 2007
programmer 	oscat
tested by	oscat

Pulse_length indicates on 3 outputs if an input pulse had been shorter than T_short (short = True), longer than T_long (long = True) or between T_short and T_long (middle = True).

*)

(* read system time *)
tx := DWORD_TO_TIME(OSCAT_BASIC.T_PLC_MS());

(* reset outputs, they should only be active 1 cycle *)
short := FALSE;
Middle := FALSE;
long := FALSE;

(* detect rising edge *)
IF in AND NOT edge THEN
	edge := TRUE;
	tn := tx;

(* detect for falling edge *)
ELSIF NOT in AND edge THEN
	edge := FALSE;
	tn := tx - tn;
	IF tn < t_short THEN
		short := TRUE;
	ELSIF tn > t_long THEN
		long := TRUE;
	ELSE
		Middle := TRUE;
	END_IF;

(* generate long pulse as soon as T_long is reached *)
ELSIF in AND tx - tn > t_long THEN
	long := TRUE;
END_IF;


(* revision history

hm	15. feb 2006	rev 1.0
	original version

hm	15 sep 2007		rev 1.1
	replaced Time() with T_PLC_MS for compatibility and performance reasons

*)

END_FUNCTION_BLOCK

// POUs/electrical/PULSE_T
FUNCTION_BLOCK PULSE_T
VAR_INPUT
	IN : BOOL;
	T1 : TIME;
	T2 : TIME;
	RST : BOOL;
END_VAR
VAR_OUTPUT
	Q : BOOL;
END_VAR
VAR
	init: BOOL;
	last: TIME;
	tx: TIME;
	edge: BOOL;
END_VAR


(*
version 1.0	15. jul. 2008
programmer 	hugo
tested by	oscat

PULSE_T generates a pulse of length T2 if the input pulse is shorter than T1.
if the input pulse is longer than T1, the output follows the input.
and rising edge on in will kill a possible output pulse and generate a new pulse instead.

*)

tx := DWORD_TO_TIME(OSCAT_BASIC.T_PLC_MS());
IF NOT init THEN
	init := TRUE;
	last := tx;
ELSIF RST THEN
	(* asynchronous reset *)
	Q := FALSE;
ELSIF IN AND NOT edge AND NOT Q THEN
	(* a rising edge on in will reversre the output status, if new pulse is startet the start time is stored in last *)
	last := tx;
	Q := TRUE;
ELSIF NOT IN AND edge AND ((tx - last) > T1) THEN
	(* a falling edge on IN will clear the output if in was high for more then T1 *)
	Q := FALSE;
ELSIF (tx - last) >= T2 THEN
	(* timeout for long pulse if second click did not occur or in stays high *)
	Q := FALSE;
END_IF;

edge := IN;

(* revision histroy
hm	15. jul. 2008	rev 1.0
	original release


*)

END_FUNCTION_BLOCK

// POUs/HLK/SDD_NH3
FUNCTION SDD_NH3 : REAL
VAR_INPUT
	T : REAL;
END_VAR


(*
version 1.0	19 Aug 2009
programmer 	hugo
tested by		tobias

this function calculates the vapor saturation pressure for NH3 gas
valid input temperature range is -109°C .. 98 °C

*)

(*
calculate according to NIST
Antoine Equation Parameters
log10(P) = A - (B / (T + C))
	P = vapor pressure (bar)
	T = temperature (K)
Temperature (K)	A	B	C	Reference	Comment

 T = 164.0 - 239.5, A =	3.18757, B =506.713, C=-80.78	Stull, 1947	Coefficents calculated by NIST from author's data.
 T = 239.5 - 371.4, A =	4.86886, B = 1113.928, C = -10.409	Stull, 1947	Coefficents calculated by NIST from author's data.
*)



IF T < -33.65 THEN
	SDD_NH3 := EXP(7.3396511649 - ( 1166.7498002 / ( T + 192.37 )));
ELSE
	SDD_NH3 := EXP(11.210964456 - ( 2564.9140075 / ( T + 262.741 )));
END_IF;



(* revision history

hm 19 aug 2009		rev 1.0
	original version

*)

END_FUNCTION

// POUs/HLK/SDT_NH3
FUNCTION SDT_NH3 : REAL
VAR_INPUT
	P : REAL;
END_VAR


(*
version 1.0	20 Aug 2009
programmer 	hugo
tested by		tobias

this function calculates the vapor saturation temperature for NH3 gas
valid input pressure is 0.001 bar .. 60 bar.

*)

(*
calculate according to NIST
Antoine Equation Parameters
log10(P) = A - (B / (T + C))
	P = vapor pressure (bar)
	T = temperature (K)
Temperature (K)	A	B	C	Reference	Comment

 T = 164.0 - 239.5, A =	3.18757, B =506.713, C=-80.78	Stull, 1947	Coefficents calculated by NIST from author's data.
 T = 239.5 - 371.4, A =	4.86886, B = 1113.928, C = -10.409	Stull, 1947	Coefficents calculated by NIST from author's data.
*)


IF P < 1.0E-3 THEN
	SDT_NH3 := -110.0;
ELSIF P < 1.0 THEN
	SDT_NH3 := 506.713 / (3.18757 - LOG(P)) - 192.37 ;
ELSE
	SDT_NH3 := 1113.928 / (4.86886 - LOG(P)) - 262.71 ;
END_IF;



(* revision history

hm 20 aug 2009		rev 1.0
	original version

*)

END_FUNCTION

// POUs/electrical/SWITCH_I
FUNCTION_BLOCK SWITCH_I
VAR_INPUT
	set : BOOL;
	in : BOOL;
	rst : BOOL;
END_VAR
VAR_INPUT CONSTANT
	T_debounce : TIME := T#10ms;
	T_reconfig : TIME := T#1s;
	T_on_max : TIME := T#0h;
END_VAR
VAR_OUTPUT
	Q : BOOL;
END_VAR
VAR
	state : BYTE;
	edge : BOOL;
	r_edge : BOOL;
	T_on : TIME;
	tx: TIME;
END_VAR

(*
version 1.1	15 sep 2007
programmer 	oscat
tested by	oscat

this is an intelligent switch interface which has an autodetect feature for in and it will detect the type of switch connected automatically
the input can be connected to low active pulses, high active pulses and on/off switch.
it will automatically adjust to the correct type without manual adjustment
a configurable debounce timer will debounce input signals
if t_on_max is set to anything other then 0 the output will be turned off after the max on time is reached.

*)

(* read system time *)
tx := DWORD_TO_TIME(OSCAT_BASIC.T_PLC_MS());

(* asynchronous set and reset first *)
IF set AND NOT rst THEN
	Q := TRUE;
	T_on := tx;
ELSIF rst THEN
	Q := FALSE;
(* check FOR input edge AND start debounce timer *)
ELSIF (in XOR edge) AND NOT (state = 1) THEN
	state := 1;
	T_on := Tx;
(* edge was detected and debounce time elapsed *)
ELSIF (state = 1) AND (Tx - t_debounce >= T_on) THEN
	state := 2;
	(* react on rising or falling edge depending on r_edge *)
	IF r_edge XOR in THEN Q := NOT Q; END_IF;
(* wait for T_reconfig and adjust r_edge *)
ELSIF state = 2 AND Tx - t_reconfig >= T_on THEN
	r_edge := in;
END_IF;
IF Q AND T_on_max > t#0ms AND Tx >= T_on + T_on_max THEN
	Q := FALSE;
END_IF;
edge := in;

(* revision history

hm	4 aug 2006	rev 1.0
	original version

hm	15.9.2007	rev 1.1
	replaced Time() with T_PLC_MS for compatibility and performance reasons

*)

END_FUNCTION_BLOCK

// POUs/electrical/SWITCH_X
FUNCTION_BLOCK SWITCH_X
VAR_INPUT
	IN1 : BOOL;
	IN2 : BOOL;
	IN3 : BOOL;
	IN4 : BOOL;
	IN5 : BOOL;
	IN6 : BOOL;
END_VAR
VAR_OUTPUT
	Q1 : BOOL;
	Q2 : BOOL;
	Q3 : BOOL;
	Q4 : BOOL;
	Q5 : BOOL;
	Q6 : BOOL;
	Q31 : BOOL;
	Q41 : BOOL;
	Q51 : BOOL;
	Q61 : BOOL;
	Q32 : BOOL;
	Q42 : BOOL;
	Q52 : BOOL;
	Q62 : BOOL;
END_VAR
VAR_INPUT CONSTANT
	t_debounce : TIME := t#50ms;
END_VAR
VAR
	init : BOOL;
	T1, T2, T3, T4, T5, T6 : OSCAT_BASIC.TOF;
	tx: TIME;
	x1: BOOL;
	x2: BOOL;
	E1, E2 : BOOL;
END_VAR

(*
version 1.0	15 Feb 2007
programmer 	oscat
tested by	oscat

*)

(* initialize on startup *)
IF NOT init THEN
	init := TRUE;
	IF t_debounce < t#50ms THEN tx := t#50ms; ELSE tx := t_debounce; END_IF;
	T1(PT := Tx);
	T2(PT := Tx);
	T3(PT := Tx);
	T4(PT := Tx);
	T5(PT := Tx);
	T6(PT := Tx);
ELSE
	Q1 := FALSE;
	Q2 := FALSE;
	Q3 := FALSE;
	Q4 := FALSE;
	Q5 := FALSE;
	Q6 := FALSE;
	Q31 := FALSE;
	Q41 := FALSE;
	Q51 := FALSE;
	Q61 := FALSE;
	Q32 := FALSE;
	Q42 := FALSE;
	Q52 := FALSE;
	Q62 := FALSE;
END_IF;

(* read inputs and debounce *)
	T1(IN := IN1);
	T2(IN := IN2);
	T3(IN := IN3);
	T4(IN := IN4);
	T5(IN := IN5);
	T6(IN := IN6);

(* detect edge of IN1 and IN2 *)
IF t1.Q AND NOT E1 THEN X1 := TRUE; END_IF;
IF t2.Q AND NOT E2 THEN X2 := TRUE; END_IF;

IF t1.Q THEN
	IF t3.q THEN
		q31 := TRUE;
		X1 := FALSE;
	ELSIF t4.q THEN
		q41 := TRUE;
		X1 := FALSE;
	ELSIF t5.q THEN
		q51 := TRUE;
		X1 := FALSE;
	ELSIF t6.q THEN
		q61 := TRUE;
		X1 := FALSE;
	END_IF;
ELSIF t2.Q THEN
	IF t3.q THEN
		q32 := TRUE;
		X2 := FALSE;
	ELSIF t4.q THEN
		q42 := TRUE;
		X2 := FALSE;
	ELSIF t5.q THEN
		q52 := TRUE;
		X2 := FALSE;
	ELSIF t6.q THEN
		q62 := TRUE;
		X2 := FALSE;
	END_IF;
(* in1 was active alone *)
ELSIF NOT T1.Q AND E1 AND X1 THEN
	Q1 := TRUE;
	X1 := FALSE;
ELSIF NOT T2.Q AND E2 AND X2 THEN
	Q2 := TRUE;
	X2 := FALSE;
ELSIF T3.Q THEN
	Q3 := TRUE;
ELSIF T4.Q THEN
	Q4 := TRUE;
ELSIF T5.Q THEN
	Q5 := TRUE;
ELSIF T6.Q THEN
	Q6 := TRUE;
END_IF;

(* save state of in1 and in2 *)
E1 := T1.Q;
E2 := T2.Q;

END_FUNCTION_BLOCK

// POUs/HLK/T_AVG24
FUNCTION_BLOCK T_AVG24
VAR_INPUT
	TS : INT;
	DTI : DT;
	RST : BOOL;
END_VAR
VAR_INPUT CONSTANT
	T_FILTER : TIME := T#10m;
	SCALE : REAL := 1.0;
	OFS : REAL;
END_VAR
VAR_OUTPUT
	TA : REAL;
	TP : BOOL;
END_VAR
VAR_IN_OUT
	T24 : REAL;
	T24_MAX : REAL;
	T24_MIN : REAL;
END_VAR
VAR
	samples : ARRAY[0..47] OF INT;
	pos : INT;
	init: BOOL;
	ft1 : OSCAT_BASIC.FILTER_I;
	sum : DINT;
	last: DT;
END_VAR
VAR_TEMP
	tmp_max : INT;
	tmp_min : INT;
	i: INT;
END_VAR

(*
version 1.2	13. mar. 2009
programmer 	hugo
tested by		oscat

this function calculates the averaged daytime temperature by taking 48 samples over one day.
a trigger tp will be true for one cycle when the output is updated.
using the input scale the outputs can be adjusted to different scales.

*)

(* first filter the sensor readings *)
ft1(X := TS, T := T_FILTER);

